LIN {X 0,Y 256.898,Z 678.395,A -85,B 0,C 180,E1 -18633.136,E2 -18633.136} C_VEL
LIN {X 0,Y 257.218,Z 676.163,A -85,B 0,C 180,E1 -18636.274,E2 -18636.274} C_VEL
LIN {X 0,Y 258.082,Z 673.338,A -85,B 0,C 180,E1 -18638.614,E2 -18638.614} C_VEL
LIN {X 0,Y 259.211,Z 669.508,A -85,B 0,C 180,E1 -18640.94,E2 -18640.94} C_VEL
LIN {X 0,Y 260.376,Z 664.426,A -85,B 0,C 180,E1 -18643.342,E2 -18643.342} C_VEL
LIN {X 0,Y 261.879,Z 658.391,A -85,B 0,C 180,E1 -18645.567,E2 -18645.567} C_VEL
LIN {X 0,Y 263.703,Z 650.606,A -85,B 0,C 180,E1 -18647.847,E2 -18647.847} C_VEL
LIN {X 0,Y 265.636,Z 640.929,A -85,B 0,C 180,E1 -18650.117,E2 -18650.117} C_VEL
LIN {X 0,Y 267.345,Z 631.877,A -85,B 0,C 180,E1 -18651.796,E2 -18651.796} C_VEL
LIN {X 0,Y 269.137,Z 621.362,A -85,B 0,C 180,E1 -18653.355,E2 -18653.355} C_VEL
LIN {X 0,Y 270.675,Z 609.83,A -85,B 0,C 180,E1 -18654.712,E2 -18654.712} C_VEL
LIN {X 0,Y 271.973,Z 598.532,A -85,B 0,C 180,E1 -18655.719,E2 -18655.719} C_VEL
LIN {X 0,Y 272.565,Z 586.357,A -85,B 0,C 180,E1 -18656.554,E2 -18656.554} C_VEL
LIN {X 0,Y 272.931,Z 573.758,A -85,B 0,C 180,E1 -18657.114,E2 -18657.114} C_VEL
LIN {X 0,Y 273.749,Z 534.07,A -85,B 0,C 180,E1 -18658.199,E2 -18658.199} C_VEL
LIN {X 0,Y 273.781,Z 527.785,A -85,B 0,C 180,E1 -18658.381,E2 -18658.381} C_VEL
LIN {X 0,Y 266.212,Z 511.696,A -85,B 0,C 180,E1 -18659.794,E2 -18659.794} C_VEL
LIN {X 0,Y 257.73,Z 496.288,A -85,B 0,C 180,E1 -18661.42,E2 -18661.42} C_VEL
LIN {X 0,Y 256.336,Z 493.738,A -85,B 0,C 180,E1 -18661.726,E2 -18661.726} C_VEL
LIN {X 0,Y 256.105,Z 492.716,A -85,B 0,C 180,E1 -18662.044,E2 -18662.044} C_VEL
LIN {X 0,Y 256.108,Z 492.575,A -85,B 0,C 180,E1 -18665.188,E2 -18665.188} C_VEL
LIN {X 0,Y 256.071,Z 492.587,A -85,B 0,C 180,E1 -18669.141,E2 -18669.141} C_VEL
LIN {X 0,Y 256.063,Z 492.56,A -85,B 0,C 180,E1 -18673.326,E2 -18673.326} C_VEL
LIN {X 0,Y 256.07,Z 492.567,A -85,B 0,C 180,E1 -18677.818,E2 -18677.818} C_VEL
LIN {X 0,Y 256.068,Z 492.545,A -85,B 0,C 180,E1 -18680.857,E2 -18680.857} C_VEL
LIN {X 0,Y 256.126,Z 492.571,A -85,B 0,C 180,E1 -18682.866,E2 -18682.866} C_VEL
LIN {X 0,Y 256.064,Z 492.561,A -85,B 0,C 180,E1 -18686.706,E2 -18686.706} C_VEL
LIN {X 0,Y 256.1,Z 492.529,A -85,B 0,C 180,E1 -18690.398,E2 -18690.398} C_VEL
LIN {X 0,Y 256.166,Z 492.577,A -85,B 0,C 180,E1 -18694.869,E2 -18694.869} C_VEL
LIN {X 0,Y 256.157,Z 492.568,A -85,B 0,C 180,E1 -18699.104,E2 -18699.104} C_VEL
LIN {X 0,Y 256.274,Z 492.543,A -85,B 0,C 180,E1 -18704.083,E2 -18704.083} C_VEL
LIN {X 0,Y 256.304,Z 492.547,A -85,B 0,C 180,E1 -18708.934,E2 -18708.934} C_VEL
LIN {X 0,Y 256.534,Z 492.518,A -85,B 0,C 180,E1 -18712.127,E2 -18712.127} C_VEL
LIN {X 0,Y 256.709,Z 492.489,A -85,B 0,C 180,E1 -18718.431,E2 -18718.431} C_VEL
LIN {X 0,Y 256.709,Z 492.502,A -85,B 0,C 180,E1 -18721.569,E2 -18721.569} C_VEL
LIN {X 0,Y 256.477,Z 492.531,A -85,B 0,C 180,E1 -18726.293,E2 -18726.293} C_VEL
LIN {X 0,Y 256.434,Z 492.532,A -85,B 0,C 180,E1 -18728.964,E2 -18728.964} C_VEL
LIN {X 0,Y 255.721,Z 492.619,A -85,B 0,C 180,E1 -18730.273,E2 -18730.273} C_VEL
LIN {X 0,Y 252.761,Z 492.991,A -85,B 0,C 180,E1 -18732.404,E2 -18732.404} C_VEL
LIN {X 0,Y 250.289,Z 493.308,A -85,B 0,C 180,E1 -18734.139,E2 -18734.139} C_VEL
LIN {X 0,Y 249.269,Z 493.429,A -85,B 0,C 180,E1 -18735.487,E2 -18735.487} C_VEL
LIN {X 0,Y 249.207,Z 493.429,A -85,B 0,C 180,E1 -18735.944,E2 -18735.944} C_VEL
LIN {X 0,Y 249.102,Z 493.418,A -85,B 0,C 180,E1 -18739.789,E2 -18739.789} C_VEL
LIN {X 0,Y 249.147,Z 493.434,A -85,B 0,C 180,E1 -18745.032,E2 -18745.032} C_VEL
LIN {X 0,Y 249.079,Z 493.45,A -85,B 0,C 180,E1 -18748.994,E2 -18748.994} C_VEL
LIN {X 0,Y 249.027,Z 493.446,A -85,B 0,C 180,E1 -18752.426,E2 -18752.426} C_VEL
LIN {X 0,Y 249.049,Z 493.462,A -85,B 0,C 180,E1 -18756.342,E2 -18756.342} C_VEL
LIN {X 0,Y 249.003,Z 493.47,A -85,B 0,C 180,E1 -18760.479,E2 -18760.479} C_VEL
LIN {X 0,Y 249.065,Z 493.617,A -85,B 0,C 180,E1 -18764.83,E2 -18764.83} C_VEL
LIN {X 0,Y 251.785,Z 503.076,A -85,B 0,C 180,E1 -18768.346,E2 -18768.346} C_VEL
LIN {X 0,Y 254.298,Z 513.073,A -85,B 0,C 180,E1 -18771.759,E2 -18771.759} C_VEL
LIN {X 0,Y 256.079,Z 521.057,A -85,B 0,C 180,E1 -18774.325,E2 -18774.325} C_VEL
LIN {X 0,Y 257.657,Z 529.601,A -85,B 0,C 180,E1 -18776.94,E2 -18776.94} C_VEL
LIN {X 0,Y 257.297,Z 532.64,A -85,B 0,C 180,E1 -18777.708,E2 -18777.708} C_VEL
LIN {X 0,Y 261.354,Z 564.078,A -85,B 0,C 180,E1 -18779.275,E2 -18779.275} C_VEL
LIN {X 0,Y 264.389,Z 595.733,A -85,B 0,C 180,E1 -18780.613,E2 -18780.613} C_VEL
LIN {X 0,Y 265.308,Z 609.441,A -85,B 0,C 180,E1 -18781.132,E2 -18781.132} C_VEL
LIN {X 0,Y 263.989,Z 644.739,A -85,B 0,C 180,E1 -18782.096,E2 -18782.096} C_VEL
LIN {X 0,Y 262.828,Z 658.786,A -85,B 0,C 180,E1 -18782.789,E2 -18782.789} C_VEL
LIN {X 0,Y 261.25,Z 671.74,A -85,B 0,C 180,E1 -18783.757,E2 -18783.757} C_VEL
LIN {X 0,Y 259.131,Z 683.47,A -85,B 0,C 180,E1 -18784.928,E2 -18784.928} C_VEL
LIN {X 0,Y 256.83,Z 694.835,A -85,B 0,C 180,E1 -18786.41,E2 -18786.41} C_VEL
LIN {X 0,Y 254.641,Z 705.126,A -85,B 0,C 180,E1 -18788.125,E2 -18788.125} C_VEL
LIN {X 0,Y 252.582,Z 714.429,A -85,B 0,C 180,E1 -18790.072,E2 -18790.072} C_VEL
LIN {X 0,Y 250.959,Z 722.161,A -85,B 0,C 180,E1 -18792.059,E2 -18792.059} C_VEL
LIN {X 0,Y 249.69,Z 727.412,A -85,B 0,C 180,E1 -18793.653,E2 -18793.653} C_VEL
LIN {X 0,Y 248.633,Z 734.063,A -85,B 0,C 180,E1 -18796.098,E2 -18796.098} C_VEL
LIN {X 0,Y 247.979,Z 739.385,A -85,B 0,C 180,E1 -18798.558,E2 -18798.558} C_VEL
LIN {X 0,Y 247.814,Z 743.573,A -85,B 0,C 180,E1 -18801.027,E2 -18801.027} C_VEL
LIN {X 0,Y 247.978,Z 746.708,A -85,B 0,C 180,E1 -18803.491,E2 -18803.491} C_VEL
LIN {X 0,Y 248.246,Z 748.229,A -85,B 0,C 180,E1 -18805.128,E2 -18805.128} C_VEL
LIN {X 0,Y 248.493,Z 749.321,A -85,B 0,C 180,E1 -18806.757,E2 -18806.757} C_VEL
LIN {X 0,Y 248.802,Z 750.008,A -85,B 0,C 180,E1 -18808.381,E2 -18808.381} C_VEL
LIN {X 0,Y 249.233,Z 750.293,A -85,B 0,C 180,E1 -18810,E2 -18810} C_VEL
LIN {X 0,Y 248.804,Z 750,A -85,B 0,C 180,E1 -18811.619,E2 -18811.619} C_VEL
LIN {X 0,Y 248.498,Z 749.308,A -85,B 0,C 180,E1 -18813.243,E2 -18813.243} C_VEL
LIN {X 0,Y 248.261,Z 748.212,A -85,B 0,C 180,E1 -18814.872,E2 -18814.872} C_VEL
LIN {X 0,Y 247.947,Z 745.853,A -85,B 0,C 180,E1 -18817.221,E2 -18817.221} C_VEL
LIN {X 0,Y 247.818,Z 742.225,A -85,B 0,C 180,E1 -18819.797,E2 -18819.797} C_VEL
LIN {X 0,Y 248.151,Z 737.656,A -85,B 0,C 180,E1 -18822.263,E2 -18822.263} C_VEL
LIN {X 0,Y 248.949,Z 731.901,A -85,B 0,C 180,E1 -18824.718,E2 -18824.718} C_VEL
LIN {X 0,Y 250.399,Z 724.287,A -85,B 0,C 180,E1 -18827.299,E2 -18827.299} C_VEL
LIN {X 0,Y 252.186,Z 715.948,A -85,B 0,C 180,E1 -18829.537,E2 -18829.537} C_VEL
LIN {X 0,Y 254.191,Z 706.941,A -85,B 0,C 180,E1 -18831.49,E2 -18831.49} C_VEL
LIN {X 0,Y 256.635,Z 695.91,A -85,B 0,C 180,E1 -18833.395,E2 -18833.395} C_VEL
LIN {X 0,Y 258.839,Z 684.792,A -85,B 0,C 180,E1 -18834.888,E2 -18834.888} C_VEL
LIN {X 0,Y 261.021,Z 672.375,A -85,B 0,C 180,E1 -18836.16,E2 -18836.16} C_VEL
LIN {X 0,Y 262.652,Z 659.498,A -85,B 0,C 180,E1 -18837.141,E2 -18837.141} C_VEL
LIN {X 0,Y 263.825,Z 646.314,A -85,B 0,C 180,E1 -18837.81,E2 -18837.81} C_VEL
LIN {X 0,Y 264.634,Z 624.724,A -85,B 0,C 180,E1 -18838.448,E2 -18838.448} C_VEL
LIN {X 0,Y 265.119,Z 606.949,A -85,B 0,C 180,E1 -18838.926,E2 -18838.926} C_VEL
LIN {X 0,Y 262.716,Z 577.983,A -85,B 0,C 180,E1 -18840.087,E2 -18840.087} C_VEL
LIN {X 0,Y 259.668,Z 550.828,A -85,B 0,C 180,E1 -18841.31,E2 -18841.31} C_VEL
LIN {X 0,Y 257.249,Z 532.626,A -85,B 0,C 180,E1 -18842.256,E2 -18842.256} C_VEL
LIN {X 0,Y 257.663,Z 529.472,A -85,B 0,C 180,E1 -18843.059,E2 -18843.059} C_VEL
LIN {X 0,Y 255.438,Z 518.047,A -85,B 0,C 180,E1 -18846.582,E2 -18846.582} C_VEL
LIN {X 0,Y 252.912,Z 507.399,A -85,B 0,C 180,E1 -18850.085,E2 -18850.085} C_VEL
LIN {X 0,Y 250.225,Z 497.431,A -85,B 0,C 180,E1 -18853.648,E2 -18853.648} C_VEL
LIN {X 0,Y 249.047,Z 493.501,A -85,B 0,C 180,E1 -18855.201,E2 -18855.201} C_VEL
LIN {X 0,Y 249.004,Z 493.47,A -85,B 0,C 180,E1 -18859.644,E2 -18859.644} C_VEL
LIN {X 0,Y 249.044,Z 493.462,A -85,B 0,C 180,E1 -18863.657,E2 -18863.657} C_VEL
LIN {X 0,Y 249.033,Z 493.449,A -85,B 0,C 180,E1 -18867.845,E2 -18867.845} C_VEL
LIN {X 0,Y 249.093,Z 493.441,A -85,B 0,C 180,E1 -18871.338,E2 -18871.338} C_VEL
LIN {X 0,Y 249.147,Z 493.435,A -85,B 0,C 180,E1 -18874.968,E2 -18874.968} C_VEL
LIN {X 0,Y 249.102,Z 493.417,A -85,B 0,C 180,E1 -18880.211,E2 -18880.211} C_VEL
LIN {X 0,Y 249.237,Z 493.425,A -85,B 0,C 180,E1 -18883.622,E2 -18883.622} C_VEL
LIN {X 0,Y 249.239,Z 493.419,A -85,B 0,C 180,E1 -18888.616,E2 -18888.616} C_VEL
LIN {X 0,Y 249.449,Z 493.411,A -85,B 0,C 180,E1 -18891.902,E2 -18891.902} C_VEL
LIN {X 0,Y 249.292,Z 493.41,A -85,B 0,C 180,E1 -18895.148,E2 -18895.148} C_VEL
LIN {X 0,Y 249.671,Z 493.382,A -85,B 0,C 180,E1 -18898.387,E2 -18898.387} C_VEL
LIN {X 0,Y 249.671,Z 493.368,A -85,B 0,C 180,E1 -18901.613,E2 -18901.613} C_VEL
LIN {X 0,Y 249.437,Z 493.41,A -85,B 0,C 180,E1 -18906.709,E2 -18906.709} C_VEL
LIN {X 0,Y 249.338,Z 493.403,A -85,B 0,C 180,E1 -18909.737,E2 -18909.737} C_VEL
LIN {X 0,Y 249.192,Z 493.432,A -85,B 0,C 180,E1 -18914.704,E2 -18914.704} C_VEL
LIN {X 0,Y 249.129,Z 493.447,A -85,B 0,C 180,E1 -18918.078,E2 -18918.078} C_VEL
LIN {X 0,Y 249.08,Z 493.444,A -85,B 0,C 180,E1 -18921.519,E2 -18921.519} C_VEL
LIN {X 0,Y 249.113,Z 493.454,A -85,B 0,C 180,E1 -18925.476,E2 -18925.476} C_VEL
LIN {X 0,Y 249.07,Z 493.412,A -85,B 0,C 180,E1 -18928.99,E2 -18928.99} C_VEL
LIN {X 0,Y 249.027,Z 493.417,A -85,B 0,C 180,E1 -18932.427,E2 -18932.427} C_VEL
LIN {X 0,Y 249.044,Z 493.463,A -85,B 0,C 180,E1 -18936.343,E2 -18936.343} C_VEL
LIN {X 0,Y 248.989,Z 493.424,A -85,B 0,C 180,E1 -18940.482,E2 -18940.482} C_VEL
LIN {X 0,Y 249.009,Z 493.456,A -85,B 0,C 180,E1 -18942.794,E2 -18942.794} C_VEL
LIN {X 0,Y 249.016,Z 493.434,A -85,B 0,C 180,E1 -18947.364,E2 -18947.364} C_VEL
LIN {X 0,Y 249.025,Z 493.447,A -85,B 0,C 180,E1 -18951.62,E2 -18951.62} C_VEL
LIN {X 0,Y 249.043,Z 493.376,A -85,B 0,C 180,E1 -18955.64,E2 -18955.64} C_VEL
LIN {X 0,Y 249.076,Z 493.63,A -85,B 0,C 180,E1 -18957.103,E2 -18957.103} C_VEL
LIN {X 0,Y 249.366,Z 494.727,A -85,B 0,C 180,E1 -18957.422,E2 -18957.422} C_VEL
LIN {X 0,Y 258.488,Z 511.081,A -85,B 0,C 180,E1 -18959.298,E2 -18959.298} C_VEL
LIN {X 0,Y 265.326,Z 524.858,A -85,B 0,C 180,E1 -18960.631,E2 -18960.631} C_VEL
LIN {X 0,Y 267.603,Z 530.043,A -85,B 0,C 180,E1 -18961.073,E2 -18961.073} C_VEL
LIN {X 0,Y 266.729,Z 570.85,A -85,B 0,C 180,E1 -18962.201,E2 -18962.201} C_VEL
LIN {X 0,Y 266.366,Z 584.382,A -85,B 0,C 180,E1 -18962.736,E2 -18962.736} C_VEL
LIN {X 0,Y 265.506,Z 597.64,A -85,B 0,C 180,E1 -18963.576,E2 -18963.576} C_VEL
LIN {X 0,Y 264.349,Z 609.929,A -85,B 0,C 180,E1 -18964.68,E2 -18964.68} C_VEL
LIN {X 0,Y 262.733,Z 621.407,A -85,B 0,C 180,E1 -18966.03,E2 -18966.03} C_VEL
LIN {X 0,Y 260.875,Z 632.144,A -85,B 0,C 180,E1 -18967.634,E2 -18967.634} C_VEL
LIN {X 0,Y 259.092,Z 641.336,A -85,B 0,C 180,E1 -18969.352,E2 -18969.352} C_VEL
LIN {X 0,Y 257.375,Z 649.686,A -85,B 0,C 180,E1 -18971.286,E2 -18971.286} C_VEL
LIN {X 0,Y 255.459,Z 657.796,A -85,B 0,C 180,E1 -18973.621,E2 -18973.621} C_VEL
LIN {X 0,Y 253.631,Z 664.903,A -85,B 0,C 180,E1 -18976.21,E2 -18976.21} C_VEL
LIN {X 0,Y 252.34,Z 670.272,A -85,B 0,C 180,E1 -18978.758,E2 -18978.758} C_VEL
LIN {X 0,Y 251.142,Z 674.161,A -85,B 0,C 180,E1 -18981.146,E2 -18981.146} C_VEL
LIN {X 0,Y 250.245,Z 677.03,A -85,B 0,C 180,E1 -18983.55,E2 -18983.55} C_VEL
LIN {X 0,Y 250.031,Z 678.371,A -85,B 0,C 180,E1 -18985.163,E2 -18985.163} C_VEL
LIN {X 0,Y 249.892,Z 679.322,A -85,B 0,C 180,E1 -18986.776,E2 -18986.776} C_VEL
LIN {X 0,Y 249.637,Z 680.15,A -85,B 0,C 180,E1 -18990,E2 -18990} C_VEL
LIN {X 0,Y 249.886,Z 679.382,A -85,B 0,C 180,E1 -18993.224,E2 -18993.224} C_VEL
LIN {X 0,Y 250.23,Z 677.151,A -85,B 0,C 180,E1 -18996.45,E2 -18996.45} C_VEL
LIN {X 0,Y 251.135,Z 674.326,A -85,B 0,C 180,E1 -18998.854,E2 -18998.854} C_VEL
LIN {X 0,Y 252.315,Z 670.495,A -85,B 0,C 180,E1 -19001.243,E2 -19001.243} C_VEL
LIN {X 0,Y 253.543,Z 665.412,A -85,B 0,C 180,E1 -19003.709,E2 -19003.709} C_VEL
LIN {X 0,Y 255.116,Z 659.377,A -85,B 0,C 180,E1 -19005.99,E2 -19005.99} C_VEL
LIN {X 0,Y 257.022,Z 651.591,A -85,B 0,C 180,E1 -19008.327,E2 -19008.327} C_VEL
LIN {X 0,Y 259.046,Z 641.914,A -85,B 0,C 180,E1 -19010.652,E2 -19010.652} C_VEL
LIN {X 0,Y 260.832,Z 632.861,A -85,B 0,C 180,E1 -19012.37,E2 -19012.37} C_VEL
LIN {X 0,Y 262.707,Z 622.343,A -85,B 0,C 180,E1 -19013.962,E2 -19013.962} C_VEL
LIN {X 0,Y 264.337,Z 610.656,A -85,B 0,C 180,E1 -19015.364,E2 -19015.364} C_VEL
LIN {X 0,Y 265.692,Z 599.17,A -85,B 0,C 180,E1 -19016.404,E2 -19016.404} C_VEL
LIN {X 0,Y 266.302,Z 586.905,A -85,B 0,C 180,E1 -19017.255,E2 -19017.255} C_VEL
LIN {X 0,Y 266.689,Z 574.464,A -85,B 0,C 180,E1 -19017.812,E2 -19017.812} C_VEL
LIN {X 0,Y 267.614,Z 533.588,A -85,B 0,C 180,E1 -19018.95,E2 -19018.95} C_VEL
LIN {X 0,Y 267.551,Z 529.88,A -85,B 0,C 180,E1 -19019.07,E2 -19019.07} C_VEL
LIN {X 0,Y 260.867,Z 515.53,A -85,B 0,C 180,E1 -19020.374,E2 -19020.374} C_VEL
LIN {X 0,Y 252.628,Z 500.555,A -85,B 0,C 180,E1 -19022.015,E2 -19022.015} C_VEL
LIN {X 0,Y 249.227,Z 494.41,A -85,B 0,C 180,E1 -19022.773,E2 -19022.773} C_VEL
LIN {X 0,Y 249.067,Z 493.538,A -85,B 0,C 180,E1 -19023.128,E2 -19023.128} C_VEL
LIN {X 0,Y 249.056,Z 493.44,A -85,B 0,C 180,E1 -19026.34,E2 -19026.34} C_VEL
LIN {X 0,Y 249.005,Z 493.46,A -85,B 0,C 180,E1 -19030.477,E2 -19030.477} C_VEL
LIN {X 0,Y 249.005,Z 493.459,A -85,B 0,C 180,E1 -19034.877,E2 -19034.877} C_VEL
LIN {X 0,Y 249.016,Z 493.455,A -85,B 0,C 180,E1 -19037.362,E2 -19037.362} C_VEL
LIN {X 0,Y 249.04,Z 493.438,A -85,B 0,C 180,E1 -19042.2,E2 -19042.2} C_VEL
LIN {X 0,Y 249.04,Z 493.456,A -85,B 0,C 180,E1 -19045.639,E2 -19045.639} C_VEL
LIN {X 0,Y 249.044,Z 493.401,A -85,B 0,C 180,E1 -19049.472,E2 -19049.472} C_VEL
LIN {X 0,Y 249.065,Z 493.451,A -85,B 0,C 180,E1 -19053.161,E2 -19053.161} C_VEL
LIN {X 0,Y 249.057,Z 493.448,A -85,B 0,C 180,E1 -19056.73,E2 -19056.73} C_VEL
LIN {X 0,Y 249.103,Z 493.455,A -85,B 0,C 180,E1 -19060.211,E2 -19060.211} C_VEL
LIN {X 0,Y 249.218,Z 493.421,A -85,B 0,C 180,E1 -19063.62,E2 -19063.62} C_VEL
LIN {X 0,Y 249.247,Z 493.43,A -85,B 0,C 180,E1 -19068.616,E2 -19068.616} C_VEL
LIN {X 0,Y 249.476,Z 493.394,A -85,B 0,C 180,E1 -19071.903,E2 -19071.903} C_VEL
LIN {X 0,Y 249.43,Z 493.392,A -85,B 0,C 180,E1 -19076.769,E2 -19076.769} C_VEL
LIN {X 0,Y 249.73,Z 493.374,A -85,B 0,C 180,E1 -19080,E2 -19080} C_VEL
LIN {X 0,Y 249.43,Z 493.394,A -85,B 0,C 180,E1 -19083.23,E2 -19083.23} C_VEL
LIN {X 0,Y 249.449,Z 493.408,A -85,B 0,C 180,E1 -19086.471,E2 -19086.471} C_VEL
LIN {X 0,Y 249.338,Z 493.411,A -85,B 0,C 180,E1 -19089.737,E2 -19089.737} C_VEL
LIN {X 0,Y 249.2,Z 493.443,A -85,B 0,C 180,E1 -19094.704,E2 -19094.704} C_VEL
LIN {X 0,Y 249.207,Z 493.429,A -85,B 0,C 180,E1 -19095.944,E2 -19095.944} C_VEL
LIN {X 0,Y 248.922,Z 493.461,A -85,B 0,C 180,E1 -19096.846,E2 -19096.846} C_VEL
LIN {X 0,Y 247.565,Z 493.63,A -85,B 0,C 180,E1 -19098.177,E2 -19098.177} C_VEL
LIN {X 0,Y 243.13,Z 494.189,A -85,B 0,C 180,E1 -19101.276,E2 -19101.276} C_VEL
LIN {X 0,Y 242.074,Z 494.331,A -85,B 0,C 180,E1 -19102.667,E2 -19102.667} C_VEL
LIN {X 0,Y 242.001,Z 494.333,A -85,B 0,C 180,E1 -19103.138,E2 -19103.138} C_VEL
LIN {X 0,Y 242.063,Z 494.306,A -85,B 0,C 180,E1 -19105.839,E2 -19105.839} C_VEL
LIN {X 0,Y 242.026,Z 494.335,A -85,B 0,C 180,E1 -19109.581,E2 -19109.581} C_VEL
LIN {X 0,Y 241.978,Z 494.322,A -85,B 0,C 180,E1 -19113.493,E2 -19113.493} C_VEL
LIN {X 0,Y 241.989,Z 494.328,A -85,B 0,C 180,E1 -19117.582,E2 -19117.582} C_VEL
LIN {X 0,Y 241.937,Z 494.32,A -85,B 0,C 180,E1 -19121.922,E2 -19121.922} C_VEL
LIN {X 0,Y 242.017,Z 494.458,A -85,B 0,C 180,E1 -19123.847,E2 -19123.847} C_VEL
LIN {X 0,Y 244.866,Z 504.204,A -85,B 0,C 180,E1 -19127.651,E2 -19127.651} C_VEL
LIN {X 0,Y 247.701,Z 515.638,A -85,B 0,C 180,E1 -19131.686,E2 -19131.686} C_VEL
LIN {X 0,Y 249.66,Z 524.87,A -85,B 0,C 180,E1 -19134.722,E2 -19134.722} C_VEL
LIN {X 0,Y 250.846,Z 531.586,A -85,B 0,C 180,E1 -19136.772,E2 -19136.772} C_VEL
LIN {X 0,Y 253.162,Z 548.651,A -85,B 0,C 180,E1 -19137.709,E2 -19137.709} C_VEL
LIN {X 0,Y 256.382,Z 576.607,A -85,B 0,C 180,E1 -19139.036,E2 -19139.036} C_VEL
LIN {X 0,Y 258.761,Z 604.007,A -85,B 0,C 180,E1 -19140.193,E2 -19140.193} C_VEL
LIN {X 0,Y 258.961,Z 611.982,A -85,B 0,C 180,E1 -19140.465,E2 -19140.465} C_VEL
LIN {X 0,Y 257.728,Z 643.741,A -85,B 0,C 180,E1 -19141.355,E2 -19141.355} C_VEL
LIN {X 0,Y 256.581,Z 657.306,A -85,B 0,C 180,E1 -19142.034,E2 -19142.034} C_VEL
LIN {X 0,Y 255.017,Z 669.723,A -85,B 0,C 180,E1 -19142.954,E2 -19142.954} C_VEL
LIN {X 0,Y 253.055,Z 680.888,A -85,B 0,C 180,E1 -19144.061,E2 -19144.061} C_VEL
LIN {X 0,Y 250.628,Z 692.538,A -85,B 0,C 180,E1 -19145.569,E2 -19145.569} C_VEL
LIN {X 0,Y 248.24,Z 703.065,A -85,B 0,C 180,E1 -19147.311,E2 -19147.311} C_VEL
LIN {X 0,Y 246.28,Z 711.721,A -85,B 0,C 180,E1 -19149.102,E2 -19149.102} C_VEL
LIN {X 0,Y 244.463,Z 719.745,A -85,B 0,C 180,E1 -19151.13,E2 -19151.13} C_VEL
LIN {X 0,Y 242.599,Z 727.604,A -85,B 0,C 180,E1 -19153.594,E2 -19153.594} C_VEL
LIN {X 0,Y 241.379,Z 734.947,A -85,B 0,C 180,E1 -19156.531,E2 -19156.531} C_VEL
LIN {X 0,Y 240.814,Z 739.88,A -85,B 0,C 180,E1 -19159.065,E2 -19159.065} C_VEL
LIN {X 0,Y 240.762,Z 743.709,A -85,B 0,C 180,E1 -19161.608,E2 -19161.608} C_VEL
LIN {X 0,Y 240.915,Z 745.709,A -85,B 0,C 180,E1 -19163.299,E2 -19163.299} C_VEL
LIN {X 0,Y 241.157,Z 747.229,A -85,B 0,C 180,E1 -19164.984,E2 -19164.984} C_VEL
LIN {X 0,Y 241.433,Z 748.327,A -85,B 0,C 180,E1 -19166.662,E2 -19166.662} C_VEL
LIN {X 0,Y 241.741,Z 749.015,A -85,B 0,C 180,E1 -19168.334,E2 -19168.334} C_VEL
LIN {X 0,Y 242.193,Z 749.304,A -85,B 0,C 180,E1 -19170,E2 -19170} C_VEL
LIN {X 0,Y 241.438,Z 748.313,A -85,B 0,C 180,E1 -19173.337,E2 -19173.337} C_VEL
LIN {X 0,Y 241.194,Z 747.214,A -85,B 0,C 180,E1 -19175.015,E2 -19175.015} C_VEL
LIN {X 0,Y 240.874,Z 745.069,A -85,B 0,C 180,E1 -19177.241,E2 -19177.241} C_VEL
LIN {X 0,Y 240.772,Z 741.218,A -85,B 0,C 180,E1 -19180.086,E2 -19180.086} C_VEL
LIN {X 0,Y 241.139,Z 736.645,A -85,B 0,C 180,E1 -19182.626,E2 -19182.626} C_VEL
LIN {X 0,Y 242.025,Z 730.892,A -85,B 0,C 180,E1 -19185.15,E2 -19185.15} C_VEL
LIN {X 0,Y 243.427,Z 723.996,A -85,B 0,C 180,E1 -19187.573,E2 -19187.573} C_VEL
LIN {X 0,Y 245.094,Z 716.568,A -85,B 0,C 180,E1 -19189.689,E2 -19189.689} C_VEL
LIN {X 0,Y 247.115,Z 707.915,A -85,B 0,C 180,E1 -19191.698,E2 -19191.698} C_VEL
LIN {X 0,Y 249.579,Z 697.284,A -85,B 0,C 180,E1 -19193.657,E2 -19193.657} C_VEL
LIN {X 0,Y 252.099,Z 685.354,A -85,B 0,C 180,E1 -19195.38,E2 -19195.38} C_VEL
LIN {X 0,Y 254.357,Z 673.372,A -85,B 0,C 180,E1 -19196.679,E2 -19196.679} C_VEL
LIN {X 0,Y 256.057,Z 660.894,A -85,B 0,C 180,E1 -19197.702,E2 -19197.702} C_VEL
LIN {X 0,Y 257.397,Z 647.822,A -85,B 0,C 180,E1 -19198.444,E2 -19198.444} C_VEL
LIN {X 0,Y 258.167,Z 633.463,A -85,B 0,C 180,E1 -19198.926,E2 -19198.926} C_VEL
LIN {X 0,Y 258.835,Z 606.75,A -85,B 0,C 180,E1 -19199.671,E2 -19199.671} C_VEL
LIN {X 0,Y 256.405,Z 577.658,A -85,B 0,C 180,E1 -19200.885,E2 -19200.885} C_VEL
LIN {X 0,Y 253.501,Z 551.579,A -85,B 0,C 180,E1 -19202.104,E2 -19202.104} C_VEL
LIN {X 0,Y 250.827,Z 531.562,A -85,B 0,C 180,E1 -19203.188,E2 -19203.188} C_VEL
LIN {X 0,Y 250.082,Z 527.007,A -85,B 0,C 180,E1 -19204.553,E2 -19204.553} C_VEL
LIN {X 0,Y 248.156,Z 517.819,A -85,B 0,C 180,E1 -19207.535,E2 -19207.535} C_VEL
LIN {X 0,Y 245.987,Z 508.715,A -85,B 0,C 180,E1 -19210.661,E2 -19210.661} C_VEL
LIN {X 0,Y 243.679,Z 500.036,A -85,B 0,C 180,E1 -19213.86,E2 -19213.86} C_VEL
LIN {X 0,Y 242.014,Z 494.391,A -85,B 0,C 180,E1 -19216.152,E2 -19216.152} C_VEL
LIN {X 0,Y 241.953,Z 494.34,A -85,B 0,C 180,E1 -19220.28,E2 -19220.28} C_VEL
LIN {X 0,Y 241.984,Z 494.341,A -85,B 0,C 180,E1 -19224.489,E2 -19224.489} C_VEL
LIN {X 0,Y 241.971,Z 494.335,A -85,B 0,C 180,E1 -19228.479,E2 -19228.479} C_VEL
LIN {X 0,Y 242.004,Z 494.312,A -85,B 0,C 180,E1 -19232.312,E2 -19232.312} C_VEL
LIN {X 0,Y 242.052,Z 494.331,A -85,B 0,C 180,E1 -19236.015,E2 -19236.015} C_VEL
LIN {X 0,Y 242.03,Z 494.303,A -85,B 0,C 180,E1 -19239.607,E2 -19239.607} C_VEL
LIN {X 0,Y 242.159,Z 494.299,A -85,B 0,C 180,E1 -19243.278,E2 -19243.278} C_VEL
LIN {X 0,Y 242.175,Z 494.299,A -85,B 0,C 180,E1 -19248.279,E2 -19248.279} C_VEL
LIN {X 0,Y 242.395,Z 494.29,A -85,B 0,C 180,E1 -19251.665,E2 -19251.665} C_VEL
LIN {X 0,Y 242.252,Z 494.287,A -85,B 0,C 180,E1 -19255.007,E2 -19255.007} C_VEL
LIN {X 0,Y 242.631,Z 494.259,A -85,B 0,C 180,E1 -19258.34,E2 -19258.34} C_VEL
LIN {X 0,Y 242.631,Z 494.243,A -85,B 0,C 180,E1 -19261.66,E2 -19261.66} C_VEL
LIN {X 0,Y 242.418,Z 494.286,A -85,B 0,C 180,E1 -19266.681,E2 -19266.681} C_VEL
LIN {X 0,Y 242.262,Z 494.285,A -85,B 0,C 180,E1 -19270.024,E2 -19270.024} C_VEL
LIN {X 0,Y 242.151,Z 494.305,A -85,B 0,C 180,E1 -19275.142,E2 -19275.142} C_VEL
LIN {X 0,Y 242.065,Z 494.33,A -85,B 0,C 180,E1 -19278.625,E2 -19278.625} C_VEL
LIN {X 0,Y 242.002,Z 494.322,A -85,B 0,C 180,E1 -19282.181,E2 -19282.181} C_VEL
LIN {X 0,Y 242.063,Z 494.332,A -85,B 0,C 180,E1 -19285.839,E2 -19285.839} C_VEL
LIN {X 0,Y 242.004,Z 494.282,A -85,B 0,C 180,E1 -19289.584,E2 -19289.584} C_VEL
LIN {X 0,Y 241.977,Z 494.315,A -85,B 0,C 180,E1 -19293.493,E2 -19293.493} C_VEL
LIN {X 0,Y 241.986,Z 494.322,A -85,B 0,C 180,E1 -19297.583,E2 -19297.583} C_VEL
LIN {X 0,Y 241.933,Z 494.317,A -85,B 0,C 180,E1 -19301.924,E2 -19301.924} C_VEL
LIN {X 0,Y 241.935,Z 494.318,A -85,B 0,C 180,E1 -19306.572,E2 -19306.572} C_VEL
LIN {X 0,Y 241.955,Z 494.347,A -85,B 0,C 180,E1 -19310.282,E2 -19310.282} C_VEL
LIN {X 0,Y 241.981,Z 494.258,A -85,B 0,C 180,E1 -19314.489,E2 -19314.489} C_VEL
LIN {X 0,Y 242.053,Z 494.601,A -85,B 0,C 180,E1 -19316.082,E2 -19316.082} C_VEL
LIN {X 0,Y 242.36,Z 495.793,A -85,B 0,C 180,E1 -19316.359,E2 -19316.359} C_VEL
LIN {X 0,Y 251.819,Z 512.356,A -85,B 0,C 180,E1 -19318.398,E2 -19318.398} C_VEL
LIN {X 0,Y 259.348,Z 527.313,A -85,B 0,C 180,E1 -19319.931,E2 -19319.931} C_VEL
LIN {X 0,Y 261.396,Z 532.057,A -85,B 0,C 180,E1 -19320.35,E2 -19320.35} C_VEL
LIN {X 0,Y 260.534,Z 573.012,A -85,B 0,C 180,E1 -19321.516,E2 -19321.516} C_VEL
LIN {X 0,Y 260.13,Z 586.272,A -85,B 0,C 180,E1 -19322.08,E2 -19322.08} C_VEL
LIN {X 0,Y 259.225,Z 598.638,A -85,B 0,C 180,E1 -19322.884,E2 -19322.884} C_VEL
LIN {X 0,Y 258.014,Z 610.923,A -85,B 0,C 180,E1 -19324.012,E2 -19324.012} C_VEL
LIN {X 0,Y 256.332,Z 622.398,A -85,B 0,C 180,E1 -19325.392,E2 -19325.392} C_VEL
LIN {X 0,Y 254.39,Z 633.136,A -85,B 0,C 180,E1 -19327.032,E2 -19327.032} C_VEL
LIN {X 0,Y 252.527,Z 642.328,A -85,B 0,C 180,E1 -19328.79,E2 -19328.79} C_VEL
LIN {X 0,Y 250.728,Z 650.677,A -85,B 0,C 180,E1 -19330.771,E2 -19330.771} C_VEL
LIN {X 0,Y 248.724,Z 658.787,A -85,B 0,C 180,E1 -19333.165,E2 -19333.165} C_VEL
LIN {X 0,Y 246.812,Z 665.893,A -85,B 0,C 180,E1 -19335.821,E2 -19335.821} C_VEL
LIN {X 0,Y 245.451,Z 671.262,A -85,B 0,C 180,E1 -19338.438,E2 -19338.438} C_VEL
LIN {X 0,Y 244.2,Z 675.15,A -85,B 0,C 180,E1 -19340.893,E2 -19340.893} C_VEL
LIN {X 0,Y 243.26,Z 678.019,A -85,B 0,C 180,E1 -19343.364,E2 -19343.364} C_VEL
LIN {X 0,Y 243.028,Z 679.36,A -85,B 0,C 180,E1 -19345.023,E2 -19345.023} C_VEL
LIN {X 0,Y 242.879,Z 680.31,A -85,B 0,C 180,E1 -19346.682,E2 -19346.682} C_VEL
LIN {X 0,Y 242.61,Z 681.138,A -85,B 0,C 180,E1 -19350,E2 -19350} C_VEL
LIN {X 0,Y 242.873,Z 680.369,A -85,B 0,C 180,E1 -19353.318,E2 -19353.318} C_VEL
LIN {X 0,Y 243.245,Z 678.138,A -85,B 0,C 180,E1 -19356.636,E2 -19356.636} C_VEL
LIN {X 0,Y 244.193,Z 675.313,A -85,B 0,C 180,E1 -19359.108,E2 -19359.108} C_VEL
LIN {X 0,Y 245.425,Z 671.482,A -85,B 0,C 180,E1 -19361.563,E2 -19361.563} C_VEL
LIN {X 0,Y 246.721,Z 666.399,A -85,B 0,C 180,E1 -19364.095,E2 -19364.095} C_VEL
LIN {X 0,Y 248.367,Z 660.363,A -85,B 0,C 180,E1 -19366.437,E2 -19366.437} C_VEL
LIN {X 0,Y 250.36,Z 652.577,A -85,B 0,C 180,E1 -19368.833,E2 -19368.833} C_VEL
LIN {X 0,Y 252.48,Z 642.9,A -85,B 0,C 180,E1 -19371.214,E2 -19371.214} C_VEL
LIN {X 0,Y 254.348,Z 633.845,A -85,B 0,C 180,E1 -19372.972,E2 -19372.972} C_VEL
LIN {X 0,Y 256.301,Z 623.326,A -85,B 0,C 180,E1 -19374.6,E2 -19374.6} C_VEL
LIN {X 0,Y 258.007,Z 611.638,A -85,B 0,C 180,E1 -19376.032,E2 -19376.032} C_VEL
LIN {X 0,Y 259.412,Z 600.151,A -85,B 0,C 180,E1 -19377.095,E2 -19377.095} C_VEL
LIN {X 0,Y 260.082,Z 587.515,A -85,B 0,C 180,E1 -19377.985,E2 -19377.985} C_VEL
LIN {X 0,Y 260.489,Z 575.314,A -85,B 0,C 180,E1 -19378.538,E2 -19378.538} C_VEL
LIN {X 0,Y 261.455,Z 534.264,A -85,B 0,C 180,E1 -19379.708,E2 -19379.708} C_VEL
LIN {X 0,Y 261.41,Z 531.937,A -85,B 0,C 180,E1 -19379.787,E2 -19379.787} C_VEL
LIN {X 0,Y 254.491,Z 517.288,A -85,B 0,C 180,E1 -19381.195,E2 -19381.195} C_VEL
LIN {X 0,Y 245.744,Z 501.586,A -85,B 0,C 180,E1 -19383.027,E2 -19383.027} C_VEL
LIN {X 0,Y 243.114,Z 497.349,A -85,B 0,C 180,E1 -19383.595,E2 -19383.595} C_VEL
LIN {X 0,Y 242.134,Z 494.974,A -85,B 0,C 180,E1 -19383.934,E2 -19383.934} C_VEL
LIN {X 0,Y 242.022,Z 494.377,A -85,B 0,C 180,E1 -19384.368,E2 -19384.368} C_VEL
LIN {X 0,Y 241.995,Z 494.327,A -85,B 0,C 180,E1 -19388.359,E2 -19388.359} C_VEL
LIN {X 0,Y 241.937,Z 494.319,A -85,B 0,C 180,E1 -19391.921,E2 -19391.921} C_VEL
LIN {X 0,Y 241.935,Z 494.349,A -85,B 0,C 180,E1 -19396.57,E2 -19396.57} C_VEL
LIN {X 0,Y 241.992,Z 494.305,A -85,B 0,C 180,E1 -19401.639,E2 -19401.639} C_VEL
LIN {X 0,Y 241.984,Z 494.343,A -85,B 0,C 180,E1 -19404.488,E2 -19404.488} C_VEL
LIN {X 0,Y 241.969,Z 494.285,A -85,B 0,C 180,E1 -19408.479,E2 -19408.479} C_VEL
LIN {X 0,Y 241.997,Z 494.315,A -85,B 0,C 180,E1 -19412.311,E2 -19412.311} C_VEL
LIN {X 0,Y 242.037,Z 494.33,A -85,B 0,C 180,E1 -19416.014,E2 -19416.014} C_VEL
LIN {X 0,Y 242.031,Z 494.332,A -85,B 0,C 180,E1 -19419.607,E2 -19419.607} C_VEL
LIN {X 0,Y 242.159,Z 494.302,A -85,B 0,C 180,E1 -19423.278,E2 -19423.278} C_VEL
LIN {X 0,Y 242.181,Z 494.314,A -85,B 0,C 180,E1 -19428.279,E2 -19428.279} C_VEL
LIN {X 0,Y 242.423,Z 494.269,A -85,B 0,C 180,E1 -19431.665,E2 -19431.665} C_VEL
LIN {X 0,Y 242.255,Z 494.302,A -85,B 0,C 180,E1 -19435.007,E2 -19435.007} C_VEL
LIN {X 0,Y 242.631,Z 494.241,A -85,B 0,C 180,E1 -19438.34,E2 -19438.34} C_VEL
LIN {X 0,Y 242.631,Z 494.255,A -85,B 0,C 180,E1 -19441.66,E2 -19441.66} C_VEL
LIN {X 0,Y 242.419,Z 494.284,A -85,B 0,C 180,E1 -19446.659,E2 -19446.659} C_VEL
LIN {X 0,Y 242.262,Z 494.29,A -85,B 0,C 180,E1 -19450.024,E2 -19450.024} C_VEL
LIN {X 0,Y 242.162,Z 494.318,A -85,B 0,C 180,E1 -19455.141,E2 -19455.141} C_VEL
LIN {X 0,Y 242.066,Z 494.289,A -85,B 0,C 180,E1 -19458.625,E2 -19458.625} C_VEL
LIN {X 0,Y 242.001,Z 494.333,A -85,B 0,C 180,E1 -19463.138,E2 -19463.138} C_VEL
LIN {X 0,Y 241.369,Z 494.415,A -85,B 0,C 180,E1 -19464.526,E2 -19464.526} C_VEL
LIN {X 0,Y 238.53,Z 494.768,A -85,B 0,C 180,E1 -19466.79,E2 -19466.79} C_VEL
LIN {X 0,Y 236.087,Z 495.073,A -85,B 0,C 180,E1 -19468.634,E2 -19468.634} C_VEL
LIN {X 0,Y 235.022,Z 495.212,A -85,B 0,C 180,E1 -19470.066,E2 -19470.066} C_VEL
LIN {X 0,Y 234.928,Z 495.222,A -85,B 0,C 180,E1 -19470.551,E2 -19470.551} C_VEL
LIN {X 0,Y 234.929,Z 495.208,A -85,B 0,C 180,E1 -19474.638,E2 -19474.638} C_VEL
LIN {X 0,Y 234.939,Z 495.207,A -85,B 0,C 180,E1 -19478.945,E2 -19478.945} C_VEL
LIN {X 0,Y 234.934,Z 495.37,A -85,B 0,C 180,E1 -19482.829,E2 -19482.829} C_VEL
LIN {X 0,Y 238.152,Z 506.239,A -85,B 0,C 180,E1 -19487.256,E2 -19487.256} C_VEL
LIN {X 0,Y 240.873,Z 517.324,A -85,B 0,C 180,E1 -19491.305,E2 -19491.305} C_VEL
LIN {X 0,Y 242.684,Z 525.743,A -85,B 0,C 180,E1 -19494.181,E2 -19494.181} C_VEL
LIN {X 0,Y 243.638,Z 530.582,A -85,B 0,C 180,E1 -19495.678,E2 -19495.678} C_VEL
LIN {X 0,Y 245.126,Z 534.825,A -85,B 0,C 180,E1 -19496.088,E2 -19496.088} C_VEL
LIN {X 0,Y 249.236,Z 567.218,A -85,B 0,C 180,E1 -19497.773,E2 -19497.773} C_VEL
LIN {X 0,Y 252.06,Z 598.456,A -85,B 0,C 180,E1 -19499.173,E2 -19499.173} C_VEL
LIN {X 0,Y 252.825,Z 610.698,A -85,B 0,C 180,E1 -19499.664,E2 -19499.664} C_VEL
LIN {X 0,Y 251.513,Z 642.794,A -85,B 0,C 180,E1 -19500.581,E2 -19500.581} C_VEL
LIN {X 0,Y 250.326,Z 656.442,A -85,B 0,C 180,E1 -19501.281,E2 -19501.281} C_VEL
LIN {X 0,Y 248.692,Z 668.728,A -85,B 0,C 180,E1 -19502.207,E2 -19502.207} C_VEL
LIN {X 0,Y 246.691,Z 679.895,A -85,B 0,C 180,E1 -19503.34,E2 -19503.34} C_VEL
LIN {X 0,Y 244.188,Z 691.544,A -85,B 0,C 180,E1 -19504.88,E2 -19504.88} C_VEL
LIN {X 0,Y 241.698,Z 702.069,A -85,B 0,C 180,E1 -19506.661,E2 -19506.661} C_VEL
LIN {X 0,Y 239.627,Z 710.72,A -85,B 0,C 180,E1 -19508.494,E2 -19508.494} C_VEL
LIN {X 0,Y 237.691,Z 718.739,A -85,B 0,C 180,E1 -19510.572,E2 -19510.572} C_VEL
LIN {X 0,Y 235.69,Z 726.591,A -85,B 0,C 180,E1 -19513.099,E2 -19513.099} C_VEL
LIN {X 0,Y 234.741,Z 732.05,A -85,B 0,C 180,E1 -19515.257,E2 -19515.257} C_VEL
LIN {X 0,Y 233.958,Z 737.373,A -85,B 0,C 180,E1 -19517.862,E2 -19517.862} C_VEL
LIN {X 0,Y 233.672,Z 741.56,A -85,B 0,C 180,E1 -19520.479,E2 -19520.479} C_VEL
LIN {X 0,Y 233.82,Z 744.705,A -85,B 0,C 180,E1 -19523.095,E2 -19523.095} C_VEL
LIN {X 0,Y 234.075,Z 746.229,A -85,B 0,C 180,E1 -19524.832,E2 -19524.832} C_VEL
LIN {X 0,Y 234.371,Z 747.333,A -85,B 0,C 180,E1 -19526.562,E2 -19526.562} C_VEL
LIN {X 0,Y 235.153,Z 748.314,A -85,B 0,C 180,E1 -19530,E2 -19530} C_VEL
LIN {X 0,Y 234.38,Z 747.319,A -85,B 0,C 180,E1 -19533.438,E2 -19533.438} C_VEL
LIN {X 0,Y 234.108,Z 746.214,A -85,B 0,C 180,E1 -19535.167,E2 -19535.167} C_VEL
LIN {X 0,Y 233.817,Z 744.25,A -85,B 0,C 180,E1 -19537.295,E2 -19537.295} C_VEL
LIN {X 0,Y 233.707,Z 740.207,A -85,B 0,C 180,E1 -19540.395,E2 -19540.395} C_VEL
LIN {X 0,Y 234.151,Z 735.636,A -85,B 0,C 180,E1 -19543.009,E2 -19543.009} C_VEL
LIN {X 0,Y 235.124,Z 729.884,A -85,B 0,C 180,E1 -19545.605,E2 -19545.605} C_VEL
LIN {X 0,Y 236.361,Z 723.986,A -85,B 0,C 180,E1 -19547.762,E2 -19547.762} C_VEL
LIN {X 0,Y 238.366,Z 715.559,A -85,B 0,C 180,E1 -19550.269,E2 -19550.269} C_VEL
LIN {X 0,Y 240.508,Z 706.91,A -85,B 0,C 180,E1 -19552.326,E2 -19552.326} C_VEL
LIN {X 0,Y 243.067,Z 696.278,A -85,B 0,C 180,E1 -19554.331,E2 -19554.331} C_VEL
LIN {X 0,Y 245.699,Z 684.35,A -85,B 0,C 180,E1 -19556.09,E2 -19556.09} C_VEL
LIN {X 0,Y 248.01,Z 672.364,A -85,B 0,C 180,E1 -19557.418,E2 -19557.418} C_VEL
LIN {X 0,Y 249.75,Z 659.881,A -85,B 0,C 180,E1 -19558.464,E2 -19558.464} C_VEL
LIN {X 0,Y 251.153,Z 646.732,A -85,B 0,C 180,E1 -19559.223,E2 -19559.223} C_VEL
LIN {X 0,Y 251.963,Z 631.717,A -85,B 0,C 180,E1 -19559.731,E2 -19559.731} C_VEL
LIN {X 0,Y 252.628,Z 607.74,A -85,B 0,C 180,E1 -19560.412,E2 -19560.412} C_VEL
LIN {X 0,Y 250.277,Z 578.587,A -85,B 0,C 180,E1 -19561.664,E2 -19561.664} C_VEL
LIN {X 0,Y 247.352,Z 551.751,A -85,B 0,C 180,E1 -19562.961,E2 -19562.961} C_VEL
LIN {X 0,Y 244.738,Z 533.577,A -85,B 0,C 180,E1 -19563.964,E2 -19563.964} C_VEL
LIN {X 0,Y 243.575,Z 530.216,A -85,B 0,C 180,E1 -19564.342,E2 -19564.342} C_VEL
LIN {X 0,Y 241.489,Z 520.121,A -85,B 0,C 180,E1 -19567.672,E2 -19567.672} C_VEL
LIN {X 0,Y 239.009,Z 509.591,A -85,B 0,C 180,E1 -19571.425,E2 -19571.425} C_VEL
LIN {X 0,Y 236.741,Z 501.451,A -85,B 0,C 180,E1 -19574.563,E2 -19574.563} C_VEL
LIN {X 0,Y 234.925,Z 495.303,A -85,B 0,C 180,E1 -19577.169,E2 -19577.169} C_VEL
LIN {X 0,Y 234.914,Z 495.208,A -85,B 0,C 180,E1 -19581.078,E2 -19581.078} C_VEL
LIN {X 0,Y 234.927,Z 495.208,A -85,B 0,C 180,E1 -19585.361,E2 -19585.361} C_VEL
LIN {X 0,Y 234.928,Z 495.222,A -85,B 0,C 180,E1 -19589.432,E2 -19589.432} C_VEL
LIN {X 0,Y 234.99,Z 495.184,A -85,B 0,C 180,E1 -19593.793,E2 -19593.793} C_VEL
LIN {X 0,Y 235.006,Z 495.187,A -85,B 0,C 180,E1 -19598.969,E2 -19598.969} C_VEL
LIN {X 0,Y 235.092,Z 495.175,A -85,B 0,C 180,E1 -19603.06,E2 -19603.06} C_VEL
LIN {X 0,Y 235.109,Z 495.182,A -85,B 0,C 180,E1 -19607.922,E2 -19607.922} C_VEL
LIN {X 0,Y 235.326,Z 495.17,A -85,B 0,C 180,E1 -19611.412,E2 -19611.412} C_VEL
LIN {X 0,Y 235.369,Z 495.163,A -85,B 0,C 180,E1 -19613.14,E2 -19613.14} C_VEL
LIN {X 0,Y 235.591,Z 495.135,A -85,B 0,C 180,E1 -19618.291,E2 -19618.291} C_VEL
LIN {X 0,Y 235.591,Z 495.119,A -85,B 0,C 180,E1 -19621.71,E2 -19621.71} C_VEL
LIN {X 0,Y 235.369,Z 495.162,A -85,B 0,C 180,E1 -19626.86,E2 -19626.86} C_VEL
LIN {X 0,Y 235.209,Z 495.165,A -85,B 0,C 180,E1 -19630.328,E2 -19630.328} C_VEL
LIN {X 0,Y 235.102,Z 495.179,A -85,B 0,C 180,E1 -19635.607,E2 -19635.607} C_VEL
LIN {X 0,Y 235.001,Z 495.213,A -85,B 0,C 180,E1 -19639.206,E2 -19639.206} C_VEL
LIN {X 0,Y 234.948,Z 495.201,A -85,B 0,C 180,E1 -19642.884,E2 -19642.884} C_VEL
LIN {X 0,Y 234.964,Z 495.209,A -85,B 0,C 180,E1 -19646.658,E2 -19646.658} C_VEL
LIN {X 0,Y 234.918,Z 495.158,A -85,B 0,C 180,E1 -19650.57,E2 -19650.57} C_VEL
LIN {X 0,Y 234.927,Z 495.215,A -85,B 0,C 180,E1 -19654.639,E2 -19654.639} C_VEL
LIN {X 0,Y 234.91,Z 495.18,A -85,B 0,C 180,E1 -19658.936,E2 -19658.936} C_VEL
LIN {X 0,Y 234.888,Z 495.224,A -85,B 0,C 180,E1 -19663.486,E2 -19663.486} C_VEL
LIN {X 0,Y 234.888,Z 495.196,A -85,B 0,C 180,E1 -19666.515,E2 -19666.515} C_VEL
LIN {X 0,Y 234.918,Z 495.216,A -85,B 0,C 180,E1 -19671.08,E2 -19671.08} C_VEL
LIN {X 0,Y 234.967,Z 495.314,A -85,B 0,C 180,E1 -19674.781,E2 -19674.781} C_VEL
LIN {X 0,Y 235.171,Z 496.249,A -85,B 0,C 180,E1 -19675.137,E2 -19675.137} C_VEL
LIN {X 0,Y 236.663,Z 498.982,A -85,B 0,C 180,E1 -19675.531,E2 -19675.531} C_VEL
LIN {X 0,Y 245.237,Z 513.641,A -85,B 0,C 180,E1 -19677.452,E2 -19677.452} C_VEL
LIN {X 0,Y 253.389,Z 529.799,A -85,B 0,C 180,E1 -19679.196,E2 -19679.196} C_VEL
LIN {X 0,Y 255.265,Z 534.083,A -85,B 0,C 180,E1 -19679.596,E2 -19679.596} C_VEL
LIN {X 0,Y 254.377,Z 573.098,A -85,B 0,C 180,E1 -19680.731,E2 -19680.731} C_VEL
LIN {X 0,Y 253.984,Z 585.841,A -85,B 0,C 180,E1 -19681.253,E2 -19681.253} C_VEL
LIN {X 0,Y 253.131,Z 598.344,A -85,B 0,C 180,E1 -19682.063,E2 -19682.063} C_VEL
LIN {X 0,Y 251.844,Z 610.897,A -85,B 0,C 180,E1 -19683.203,E2 -19683.203} C_VEL
LIN {X 0,Y 250.171,Z 622.33,A -85,B 0,C 180,E1 -19684.576,E2 -19684.576} C_VEL
LIN {X 0,Y 248.417,Z 631.817,A -85,B 0,C 180,E1 -19686.004,E2 -19686.004} C_VEL
LIN {X 0,Y 246.829,Z 639.476,A -85,B 0,C 180,E1 -19687.395,E2 -19687.395} C_VEL
LIN {X 0,Y 244.826,Z 648.509,A -85,B 0,C 180,E1 -19689.412,E2 -19689.412} C_VEL
LIN {X 0,Y 242.669,Z 657.265,A -85,B 0,C 180,E1 -19691.861,E2 -19691.861} C_VEL
LIN {X 0,Y 240.99,Z 663.438,A -85,B 0,C 180,E1 -19694.003,E2 -19694.003} C_VEL
LIN {X 0,Y 239.451,Z 669.043,A -85,B 0,C 180,E1 -19696.42,E2 -19696.42} C_VEL
LIN {X 0,Y 238.052,Z 673.651,A -85,B 0,C 180,E1 -19698.937,E2 -19698.937} C_VEL
LIN {X 0,Y 236.866,Z 677.187,A -85,B 0,C 180,E1 -19701.469,E2 -19701.469} C_VEL
LIN {X 0,Y 236.278,Z 679.008,A -85,B 0,C 180,E1 -19703.167,E2 -19703.167} C_VEL
LIN {X 0,Y 236.026,Z 680.349,A -85,B 0,C 180,E1 -19704.875,E2 -19704.875} C_VEL
LIN {X 0,Y 235.866,Z 681.298,A -85,B 0,C 180,E1 -19706.584,E2 -19706.584} C_VEL
LIN {X 0,Y 235.582,Z 682.126,A -85,B 0,C 180,E1 -19710,E2 -19710} C_VEL
LIN {X 0,Y 235.861,Z 681.357,A -85,B 0,C 180,E1 -19713.416,E2 -19713.416} C_VEL
LIN {X 0,Y 236.263,Z 679.126,A -85,B 0,C 180,E1 -19716.833,E2 -19716.833} C_VEL
LIN {X 0,Y 237.256,Z 676.3,A -85,B 0,C 180,E1 -19719.376,E2 -19719.376} C_VEL
LIN {X 0,Y 238.544,Z 672.469,A -85,B 0,C 180,E1 -19721.901,E2 -19721.901} C_VEL
LIN {X 0,Y 239.91,Z 667.385,A -85,B 0,C 180,E1 -19724.504,E2 -19724.504} C_VEL
LIN {X 0,Y 241.634,Z 661.349,A -85,B 0,C 180,E1 -19726.909,E2 -19726.909} C_VEL
LIN {X 0,Y 243.718,Z 653.563,A -85,B 0,C 180,E1 -19729.367,E2 -19729.367} C_VEL
LIN {X 0,Y 245.94,Z 643.885,A -85,B 0,C 180,E1 -19731.807,E2 -19731.807} C_VEL
LIN {X 0,Y 247.892,Z 634.83,A -85,B 0,C 180,E1 -19733.606,E2 -19733.606} C_VEL
LIN {X 0,Y 249.92,Z 624.312,A -85,B 0,C 180,E1 -19735.271,E2 -19735.271} C_VEL
LIN {X 0,Y 251.711,Z 612.62,A -85,B 0,C 180,E1 -19736.735,E2 -19736.735} C_VEL
LIN {X 0,Y 253.17,Z 601.132,A -85,B 0,C 180,E1 -19737.82,E2 -19737.82} C_VEL
LIN {X 0,Y 253.91,Z 588.8,A -85,B 0,C 180,E1 -19738.708,E2 -19738.708} C_VEL
LIN {X 0,Y 254.324,Z 575.94,A -85,B 0,C 180,E1 -19739.31,E2 -19739.31} C_VEL
LIN {X 0,Y 255.272,Z 533.889,A -85,B 0,C 180,E1 -19740.547,E2 -19740.547} C_VEL
LIN {X 0,Y 247.85,Z 518.504,A -85,B 0,C 180,E1 -19742.124,E2 -19742.124} C_VEL
LIN {X 0,Y 238.782,Z 502.542,A -85,B 0,C 180,E1 -19744.127,E2 -19744.127} C_VEL
LIN {X 0,Y 236.41,Z 498.69,A -85,B 0,C 180,E1 -19744.673,E2 -19744.673} C_VEL
LIN {X 0,Y 235.116,Z 495.964,A -85,B 0,C 180,E1 -19745.072,E2 -19745.072} C_VEL
LIN {X 0,Y 234.987,Z 495.287,A -85,B 0,C 180,E1 -19745.413,E2 -19745.413} C_VEL
LIN {X 0,Y 234.941,Z 495.214,A -85,B 0,C 180,E1 -19748.943,E2 -19748.943} C_VEL
LIN {X 0,Y 234.888,Z 495.197,A -85,B 0,C 180,E1 -19753.485,E2 -19753.485} C_VEL
LIN {X 0,Y 234.888,Z 495.227,A -85,B 0,C 180,E1 -19756.514,E2 -19756.514} C_VEL
LIN {X 0,Y 234.915,Z 495.179,A -85,B 0,C 180,E1 -19761.078,E2 -19761.078} C_VEL
LIN {X 0,Y 234.927,Z 495.216,A -85,B 0,C 180,E1 -19765.361,E2 -19765.361} C_VEL
LIN {X 0,Y 234.918,Z 495.158,A -85,B 0,C 180,E1 -19769.43,E2 -19769.43} C_VEL
LIN {X 0,Y 234.99,Z 495.21,A -85,B 0,C 180,E1 -19773.793,E2 -19773.793} C_VEL
LIN {X 0,Y 234.993,Z 495.202,A -85,B 0,C 180,E1 -19778.968,E2 -19778.968} C_VEL
LIN {X 0,Y 235.091,Z 495.183,A -85,B 0,C 180,E1 -19783.06,E2 -19783.06} C_VEL
LIN {X 0,Y 235.141,Z 495.192,A -85,B 0,C 180,E1 -19787.923,E2 -19787.923} C_VEL
LIN {X 0,Y 235.372,Z 495.144,A -85,B 0,C 180,E1 -19791.414,E2 -19791.414} C_VEL
LIN {X 0,Y 235.399,Z 495.157,A -85,B 0,C 180,E1 -19793.141,E2 -19793.141} C_VEL
LIN {X 0,Y 235.591,Z 495.117,A -85,B 0,C 180,E1 -19798.29,E2 -19798.29} C_VEL
LIN {X 0,Y 235.591,Z 495.131,A -85,B 0,C 180,E1 -19801.709,E2 -19801.709} C_VEL
LIN {X 0,Y 235.369,Z 495.162,A -85,B 0,C 180,E1 -19806.86,E2 -19806.86} C_VEL
LIN {X 0,Y 235.209,Z 495.166,A -85,B 0,C 180,E1 -19810.328,E2 -19810.328} C_VEL
LIN {X 0,Y 235.109,Z 495.192,A -85,B 0,C 180,E1 -19815.607,E2 -19815.607} C_VEL
LIN {X 0,Y 235.002,Z 495.169,A -85,B 0,C 180,E1 -19819.206,E2 -19819.206} C_VEL
LIN {X 0,Y 234.945,Z 495.216,A -85,B 0,C 180,E1 -19823.124,E2 -19823.124} C_VEL
LIN {X 0,Y 234.966,Z 495.185,A -85,B 0,C 180,E1 -19826.658,E2 -19826.658} C_VEL
LIN {X 0,Y 234.928,Z 495.222,A -85,B 0,C 180,E1 -19830.551,E2 -19830.551} C_VEL
LIN {X 0,Y 234.246,Z 495.309,A -85,B 0,C 180,E1 -19831.981,E2 -19831.981} C_VEL
LIN {X 0,Y 231.407,Z 495.657,A -85,B 0,C 180,E1 -19834.315,E2 -19834.315} C_VEL
LIN {X 0,Y 228.991,Z 495.961,A -85,B 0,C 180,E1 -19836.217,E2 -19836.217} C_VEL
LIN {X 0,Y 227.935,Z 496.078,A -85,B 0,C 180,E1 -19837.693,E2 -19837.693} C_VEL
LIN {X 0,Y 227.837,Z 496.088,A -85,B 0,C 180,E1 -19838.193,E2 -19838.193} C_VEL
LIN {X 0,Y 227.867,Z 496.292,A -85,B 0,C 180,E1 -19841.742,E2 -19841.742} C_VEL
LIN {X 0,Y 230.713,Z 505.796,A -85,B 0,C 180,E1 -19845.837,E2 -19845.837} C_VEL
LIN {X 0,Y 233.154,Z 515.092,A -85,B 0,C 180,E1 -19849.465,E2 -19849.465} C_VEL
LIN {X 0,Y 235.744,Z 526.581,A -85,B 0,C 180,E1 -19853.603,E2 -19853.603} C_VEL
LIN {X 0,Y 236.274,Z 529.34,A -85,B 0,C 180,E1 -19854.449,E2 -19854.449} C_VEL
LIN {X 0,Y 239.397,Z 537.403,A -85,B 0,C 180,E1 -19855.286,E2 -19855.286} C_VEL
LIN {X 0,Y 243.361,Z 569.807,A -85,B 0,C 180,E1 -19857.018,E2 -19857.018} C_VEL
LIN {X 0,Y 246.355,Z 604.403,A -85,B 0,C 180,E1 -19858.605,E2 -19858.605} C_VEL
LIN {X 0,Y 246.592,Z 612.294,A -85,B 0,C 180,E1 -19858.898,E2 -19858.898} C_VEL
LIN {X 0,Y 245.317,Z 641.982,A -85,B 0,C 180,E1 -19859.771,E2 -19859.771} C_VEL
LIN {X 0,Y 244.057,Z 655.576,A -85,B 0,C 180,E1 -19860.481,E2 -19860.481} C_VEL
LIN {X 0,Y 242.405,Z 667.731,A -85,B 0,C 180,E1 -19861.421,E2 -19861.421} C_VEL
LIN {X 0,Y 240.344,Z 678.898,A -85,B 0,C 180,E1 -19862.578,E2 -19862.578} C_VEL
LIN {X 0,Y 237.745,Z 690.545,A -85,B 0,C 180,E1 -19864.15,E2 -19864.15} C_VEL
LIN {X 0,Y 235.481,Z 699.994,A -85,B 0,C 180,E1 -19865.772,E2 -19865.772} C_VEL
LIN {X 0,Y 232.982,Z 709.717,A -85,B 0,C 180,E1 -19867.848,E2 -19867.848} C_VEL
LIN {X 0,Y 230.937,Z 717.732,A -85,B 0,C 180,E1 -19869.979,E2 -19869.979} C_VEL
LIN {X 0,Y 229.117,Z 724.391,A -85,B 0,C 180,E1 -19872.137,E2 -19872.137} C_VEL
LIN {X 0,Y 227.826,Z 731.045,A -85,B 0,C 180,E1 -19874.799,E2 -19874.799} C_VEL
LIN {X 0,Y 226.937,Z 736.364,A -85,B 0,C 180,E1 -19877.48,E2 -19877.48} C_VEL
LIN {X 0,Y 226.607,Z 740.553,A -85,B 0,C 180,E1 -19880.179,E2 -19880.179} C_VEL
LIN {X 0,Y 226.754,Z 743.705,A -85,B 0,C 180,E1 -19882.879,E2 -19882.879} C_VEL
LIN {X 0,Y 226.975,Z 745.228,A -85,B 0,C 180,E1 -19884.67,E2 -19884.67} C_VEL
LIN {X 0,Y 227.309,Z 746.338,A -85,B 0,C 180,E1 -19886.455,E2 -19886.455} C_VEL
LIN {X 0,Y 228.111,Z 747.324,A -85,B 0,C 180,E1 -19890,E2 -19890} C_VEL
LIN {X 0,Y 227.32,Z 746.324,A -85,B 0,C 180,E1 -19893.545,E2 -19893.545} C_VEL
LIN {X 0,Y 227.025,Z 745.213,A -85,B 0,C 180,E1 -19895.329,E2 -19895.329} C_VEL
LIN {X 0,Y 226.746,Z 743.462,A -85,B 0,C 180,E1 -19897.323,E2 -19897.323} C_VEL
LIN {X 0,Y 226.673,Z 739.2,A -85,B 0,C 180,E1 -19900.721,E2 -19900.721} C_VEL
LIN {X 0,Y 227.184,Z 734.628,A -85,B 0,C 180,E1 -19903.415,E2 -19903.415} C_VEL
LIN {X 0,Y 228.243,Z 728.876,A -85,B 0,C 180,E1 -19906.088,E2 -19906.088} C_VEL
LIN {X 0,Y 229.761,Z 722.369,A -85,B 0,C 180,E1 -19908.515,E2 -19908.515} C_VEL
LIN {X 0,Y 231.684,Z 714.554,A -85,B 0,C 180,E1 -19910.881,E2 -19910.881} C_VEL
LIN {X 0,Y 233.918,Z 705.903,A -85,B 0,C 180,E1 -19912.99,E2 -19912.99} C_VEL
LIN {X 0,Y 236.531,Z 695.264,A -85,B 0,C 180,E1 -19915.049,E2 -19915.049} C_VEL
LIN {X 0,Y 239.349,Z 683.348,A -85,B 0,C 180,E1 -19916.836,E2 -19916.836} C_VEL
LIN {X 0,Y 241.709,Z 671.356,A -85,B 0,C 180,E1 -19918.195,E2 -19918.195} C_VEL
LIN {X 0,Y 243.517,Z 658.872,A -85,B 0,C 180,E1 -19919.262,E2 -19919.262} C_VEL
LIN {X 0,Y 244.998,Z 645.741,A -85,B 0,C 180,E1 -19920.03,E2 -19920.03} C_VEL
LIN {X 0,Y 245.784,Z 630.775,A -85,B 0,C 180,E1 -19920.554,E2 -19920.554} C_VEL
LIN {X 0,Y 246.479,Z 608.517,A -85,B 0,C 180,E1 -19921.195,E2 -19921.195} C_VEL
LIN {X 0,Y 243.891,Z 575.826,A -85,B 0,C 180,E1 -19922.65,E2 -19922.65} C_VEL
LIN {X 0,Y 240.383,Z 545.459,A -85,B 0,C 180,E1 -19924.223,E2 -19924.223} C_VEL
LIN {X 0,Y 238.949,Z 535.997,A -85,B 0,C 180,E1 -19924.782,E2 -19924.782} C_VEL
LIN {X 0,Y 236.221,Z 529.098,A -85,B 0,C 180,E1 -19925.542,E2 -19925.542} C_VEL
LIN {X 0,Y 233.775,Z 517.691,A -85,B 0,C 180,E1 -19929.515,E2 -19929.515} C_VEL
LIN {X 0,Y 231.012,Z 506.81,A -85,B 0,C 180,E1 -19933.675,E2 -19933.675} C_VEL
LIN {X 0,Y 228.402,Z 498.003,A -85,B 0,C 180,E1 -19937.394,E2 -19937.394} C_VEL
LIN {X 0,Y 227.869,Z 496.194,A -85,B 0,C 180,E1 -19938.267,E2 -19938.267} C_VEL
LIN {X 0,Y 227.888,Z 496.092,A -85,B 0,C 180,E1 -19943.304,E2 -19943.304} C_VEL
LIN {X 0,Y 227.876,Z 496.078,A -85,B 0,C 180,E1 -19946.377,E2 -19946.377} C_VEL
LIN {X 0,Y 227.915,Z 496.092,A -85,B 0,C 180,E1 -19950.437,E2 -19950.437} C_VEL
LIN {X 0,Y 227.924,Z 496.069,A -85,B 0,C 180,E1 -19954.425,E2 -19954.425} C_VEL
LIN {X 0,Y 227.957,Z 496.078,A -85,B 0,C 180,E1 -19958.287,E2 -19958.287} C_VEL
LIN {X 0,Y 228.03,Z 496.05,A -85,B 0,C 180,E1 -19962.826,E2 -19962.826} C_VEL
LIN {X 0,Y 228.067,Z 496.062,A -85,B 0,C 180,E1 -19967.543,E2 -19967.543} C_VEL
LIN {X 0,Y 228.263,Z 496.047,A -85,B 0,C 180,E1 -19971.144,E2 -19971.144} C_VEL
LIN {X 0,Y 228.319,Z 496.042,A -85,B 0,C 180,E1 -19972.928,E2 -19972.928} C_VEL
LIN {X 0,Y 228.549,Z 496.012,A -85,B 0,C 180,E1 -19978.238,E2 -19978.238} C_VEL
LIN {X 0,Y 228.55,Z 495.995,A -85,B 0,C 180,E1 -19981.762,E2 -19981.762} C_VEL
LIN {X 0,Y 228.32,Z 496.039,A -85,B 0,C 180,E1 -19987.073,E2 -19987.073} C_VEL
LIN {X 0,Y 228.141,Z 496.048,A -85,B 0,C 180,E1 -19990.652,E2 -19990.652} C_VEL
LIN {X 0,Y 228.055,Z 496.068,A -85,B 0,C 180,E1 -19994.273,E2 -19994.273} C_VEL
LIN {X 0,Y 227.998,Z 496.077,A -85,B 0,C 180,E1 -19997.954,E2 -19997.954} C_VEL
LIN {X 0,Y 227.912,Z 496.076,A -85,B 0,C 180,E1 -20002.321,E2 -20002.321} C_VEL
LIN {X 0,Y 227.938,Z 496.084,A -85,B 0,C 180,E1 -20006.603,E2 -20006.603} C_VEL
LIN {X 0,Y 227.893,Z 496.032,A -85,B 0,C 180,E1 -20010.291,E2 -20010.291} C_VEL
LIN {X 0,Y 227.874,Z 496.073,A -85,B 0,C 180,E1 -20013.721,E2 -20013.721} C_VEL
LIN {X 0,Y 227.841,Z 496.071,A -85,B 0,C 180,E1 -20018.092,E2 -20018.092} C_VEL
LIN {X 0,Y 227.808,Z 496.09,A -85,B 0,C 180,E1 -20022.743,E2 -20022.743} C_VEL
LIN {X 0,Y 227.834,Z 496.091,A -85,B 0,C 180,E1 -20025.193,E2 -20025.193} C_VEL
LIN {X 0,Y 227.825,Z 496.093,A -85,B 0,C 180,E1 -20029.624,E2 -20029.624} C_VEL
LIN {X 0,Y 227.928,Z 496.217,A -85,B 0,C 180,E1 -20033.523,E2 -20033.523} C_VEL
LIN {X 0,Y 228.158,Z 497.196,A -85,B 0,C 180,E1 -20033.893,E2 -20033.893} C_VEL
LIN {X 0,Y 229.692,Z 499.931,A -85,B 0,C 180,E1 -20034.318,E2 -20034.318} C_VEL
LIN {X 0,Y 237.105,Z 512.386,A -85,B 0,C 180,E1 -20036.093,E2 -20036.093} C_VEL
LIN {X 0,Y 244.275,Z 525.691,A -85,B 0,C 180,E1 -20037.719,E2 -20037.719} C_VEL
LIN {X 0,Y 249.129,Z 535.995,A -85,B 0,C 180,E1 -20038.793,E2 -20038.793} C_VEL
LIN {X 0,Y 248.251,Z 574.114,A -85,B 0,C 180,E1 -20039.935,E2 -20039.935} C_VEL
LIN {X 0,Y 247.823,Z 587.2,A -85,B 0,C 180,E1 -20040.492,E2 -20040.492} C_VEL
LIN {X 0,Y 246.797,Z 600.632,A -85,B 0,C 180,E1 -20041.396,E2 -20041.396} C_VEL
LIN {X 0,Y 245.456,Z 612.911,A -85,B 0,C 180,E1 -20042.574,E2 -20042.574} C_VEL
LIN {X 0,Y 243.618,Z 624.386,A -85,B 0,C 180,E1 -20044.015,E2 -20044.015} C_VEL
LIN {X 0,Y 241.509,Z 635.121,A -85,B 0,C 180,E1 -20045.73,E2 -20045.73} C_VEL
LIN {X 0,Y 239.475,Z 644.311,A -85,B 0,C 180,E1 -20047.573,E2 -20047.573} C_VEL
LIN {X 0,Y 237.501,Z 652.659,A -85,B 0,C 180,E1 -20049.654,E2 -20049.654} C_VEL
LIN {X 0,Y 235.306,Z 660.767,A -85,B 0,C 180,E1 -20052.174,E2 -20052.174} C_VEL
LIN {X 0,Y 233.209,Z 667.872,A -85,B 0,C 180,E1 -20054.975,E2 -20054.975} C_VEL
LIN {X 0,Y 231.697,Z 673.24,A -85,B 0,C 180,E1 -20057.741,E2 -20057.741} C_VEL
LIN {X 0,Y 230.332,Z 677.128,A -85,B 0,C 180,E1 -20060.339,E2 -20060.339} C_VEL
LIN {X 0,Y 229.299,Z 679.997,A -85,B 0,C 180,E1 -20062.958,E2 -20062.958} C_VEL
LIN {X 0,Y 229.026,Z 681.337,A -85,B 0,C 180,E1 -20064.718,E2 -20064.718} C_VEL
LIN {X 0,Y 228.853,Z 682.286,A -85,B 0,C 180,E1 -20066.479,E2 -20066.479} C_VEL
LIN {X 0,Y 228.555,Z 683.114,A -85,B 0,C 180,E1 -20070,E2 -20070} C_VEL
LIN {X 0,Y 228.849,Z 682.344,A -85,B 0,C 180,E1 -20073.521,E2 -20073.521} C_VEL
LIN {X 0,Y 229.284,Z 680.114,A -85,B 0,C 180,E1 -20077.042,E2 -20077.042} C_VEL
LIN {X 0,Y 230.325,Z 677.287,A -85,B 0,C 180,E1 -20079.661,E2 -20079.661} C_VEL
LIN {X 0,Y 231.672,Z 673.456,A -85,B 0,C 180,E1 -20082.26,E2 -20082.26} C_VEL
LIN {X 0,Y 233.113,Z 668.372,A -85,B 0,C 180,E1 -20084.937,E2 -20084.937} C_VEL
LIN {X 0,Y 234.919,Z 662.335,A -85,B 0,C 180,E1 -20087.407,E2 -20087.407} C_VEL
LIN {X 0,Y 237.099,Z 654.548,A -85,B 0,C 180,E1 -20089.93,E2 -20089.93} C_VEL
LIN {X 0,Y 239.428,Z 644.87,A -85,B 0,C 180,E1 -20092.432,E2 -20092.432} C_VEL
LIN {X 0,Y 241.468,Z 635.814,A -85,B 0,C 180,E1 -20094.274,E2 -20094.274} C_VEL
LIN {X 0,Y 243.591,Z 625.293,A -85,B 0,C 180,E1 -20095.976,E2 -20095.976} C_VEL
LIN {X 0,Y 245.42,Z 613.759,A -85,B 0,C 180,E1 -20097.456,E2 -20097.456} C_VEL
LIN {X 0,Y 246.938,Z 602.455,A -85,B 0,C 180,E1 -20098.551,E2 -20098.551} C_VEL
LIN {X 0,Y 247.753,Z 590.081,A -85,B 0,C 180,E1 -20099.471,E2 -20099.471} C_VEL
LIN {X 0,Y 248.215,Z 576.743,A -85,B 0,C 180,E1 -20100.111,E2 -20100.111} C_VEL
LIN {X 0,Y 249.177,Z 535.928,A -85,B 0,C 180,E1 -20101.342,E2 -20101.342} C_VEL
LIN {X 0,Y 241.702,Z 520.652,A -85,B 0,C 180,E1 -20103.004,E2 -20103.004} C_VEL
LIN {X 0,Y 233.495,Z 506.27,A -85,B 0,C 180,E1 -20104.905,E2 -20104.905} C_VEL
LIN {X 0,Y 229.689,Z 499.958,A -85,B 0,C 180,E1 -20105.835,E2 -20105.835} C_VEL
LIN {X 0,Y 228.142,Z 497.182,A -85,B 0,C 180,E1 -20106.266,E2 -20106.266} C_VEL
LIN {X 0,Y 227.908,Z 496.16,A -85,B 0,C 180,E1 -20106.701,E2 -20106.701} C_VEL
LIN {X 0,Y 227.825,Z 496.097,A -85,B 0,C 180,E1 -20110.376,E2 -20110.376} C_VEL
LIN {X 0,Y 227.834,Z 496.098,A -85,B 0,C 180,E1 -20115.191,E2 -20115.191} C_VEL
LIN {X 0,Y 227.81,Z 496.06,A -85,B 0,C 180,E1 -20119.62,E2 -20119.62} C_VEL
LIN {X 0,Y 227.878,Z 496.1,A -85,B 0,C 180,E1 -20124.127,E2 -20124.127} C_VEL
LIN {X 0,Y 227.863,Z 496.04,A -85,B 0,C 180,E1 -20128.376,E2 -20128.376} C_VEL
LIN {X 0,Y 227.875,Z 496.074,A -85,B 0,C 180,E1 -20132.443,E2 -20132.443} C_VEL
LIN {X 0,Y 227.903,Z 496.084,A -85,B 0,C 180,E1 -20136.366,E2 -20136.366} C_VEL
LIN {X 0,Y 227.932,Z 496.092,A -85,B 0,C 180,E1 -20140.173,E2 -20140.173} C_VEL
LIN {X 0,Y 228.049,Z 496.057,A -85,B 0,C 180,E1 -20143.897,E2 -20143.897} C_VEL
LIN {X 0,Y 228.087,Z 496.073,A -85,B 0,C 180,E1 -20147.544,E2 -20147.544} C_VEL
LIN {X 0,Y 228.301,Z 496.023,A -85,B 0,C 180,E1 -20151.146,E2 -20151.146} C_VEL
LIN {X 0,Y 228.35,Z 496.034,A -85,B 0,C 180,E1 -20152.928,E2 -20152.928} C_VEL
LIN {X 0,Y 228.549,Z 495.993,A -85,B 0,C 180,E1 -20158.238,E2 -20158.238} C_VEL
LIN {X 0,Y 228.549,Z 496.008,A -85,B 0,C 180,E1 -20161.762,E2 -20161.762} C_VEL
LIN {X 0,Y 228.319,Z 496.041,A -85,B 0,C 180,E1 -20167.072,E2 -20167.072} C_VEL
LIN {X 0,Y 228.141,Z 496.044,A -85,B 0,C 180,E1 -20170.651,E2 -20170.651} C_VEL
LIN {X 0,Y 228.06,Z 496.077,A -85,B 0,C 180,E1 -20174.272,E2 -20174.272} C_VEL
LIN {X 0,Y 227.998,Z 496.044,A -85,B 0,C 180,E1 -20177.954,E2 -20177.954} C_VEL
LIN {X 0,Y 227.925,Z 496.091,A -85,B 0,C 180,E1 -20182.329,E2 -20182.329} C_VEL
LIN {X 0,Y 227.939,Z 496.06,A -85,B 0,C 180,E1 -20186.603,E2 -20186.603} C_VEL
LIN {X 0,Y 227.889,Z 496.096,A -85,B 0,C 180,E1 -20190.526,E2 -20190.526} C_VEL
LIN {X 0,Y 227.874,Z 496.078,A -85,B 0,C 180,E1 -20193.721,E2 -20193.721} C_VEL
LIN {X 0,Y 227.837,Z 496.088,A -85,B 0,C 180,E1 -20198.193,E2 -20198.193} C_VEL
LIN {X 0,Y 227.573,Z 496.409,A -85,B 0,C 180,E1 -20199.173,E2 -20199.173} C_VEL
LIN {X 0,Y 226.587,Z 497.85,A -85,B 0,C 180,E1 -20200.595,E2 -20200.595} C_VEL
LIN {X 0,Y 225.333,Z 500.11,A -85,B 0,C 180,E1 -20201.953,E2 -20201.953} C_VEL
LIN {X 0,Y 223.985,Z 503.957,A -85,B 0,C 180,E1 -20203.732,E2 -20203.732} C_VEL
LIN {X 0,Y 223.852,Z 507.084,A -85,B 0,C 180,E1 -20205.051,E2 -20205.051} C_VEL
LIN {X 0,Y 224.075,Z 508.118,A -85,B 0,C 180,E1 -20205.488,E2 -20205.488} C_VEL
LIN {X 0,Y 226.292,Z 516.514,A -85,B 0,C 180,E1 -20208.893,E2 -20208.893} C_VEL
LIN {X 0,Y 228.914,Z 528.027,A -85,B 0,C 180,E1 -20213.116,E2 -20213.116} C_VEL
LIN {X 0,Y 233.605,Z 539.657,A -85,B 0,C 180,E1 -20214.414,E2 -20214.414} C_VEL
LIN {X 0,Y 237.133,Z 568.614,A -85,B 0,C 180,E1 -20216.03,E2 -20216.03} C_VEL
LIN {X 0,Y 239.789,Z 599.668,A -85,B 0,C 180,E1 -20217.516,E2 -20217.516} C_VEL
LIN {X 0,Y 240.521,Z 611.314,A -85,B 0,C 180,E1 -20218.021,E2 -20218.021} C_VEL
LIN {X 0,Y 239.155,Z 641.206,A -85,B 0,C 180,E1 -20218.918,E2 -20218.918} C_VEL
LIN {X 0,Y 237.909,Z 654.717,A -85,B 0,C 180,E1 -20219.65,E2 -20219.65} C_VEL
LIN {X 0,Y 236.373,Z 665.621,A -85,B 0,C 180,E1 -20220.499,E2 -20220.499} C_VEL
LIN {X 0,Y 234.027,Z 677.899,A -85,B 0,C 180,E1 -20221.773,E2 -20221.773} C_VEL
LIN {X 0,Y 231.363,Z 689.549,A -85,B 0,C 180,E1 -20223.382,E2 -20223.382} C_VEL
LIN {X 0,Y 228.937,Z 698.985,A -85,B 0,C 180,E1 -20225.033,E2 -20225.033} C_VEL
LIN {X 0,Y 226.361,Z 708.712,A -85,B 0,C 180,E1 -20227.164,E2 -20227.164} C_VEL
LIN {X 0,Y 224.213,Z 716.726,A -85,B 0,C 180,E1 -20229.352,E2 -20229.352} C_VEL
LIN {X 0,Y 222.367,Z 723.394,A -85,B 0,C 180,E1 -20231.576,E2 -20231.576} C_VEL
LIN {X 0,Y 220.895,Z 730.036,A -85,B 0,C 180,E1 -20234.31,E2 -20234.31} C_VEL
LIN {X 0,Y 219.937,Z 735.356,A -85,B 0,C 180,E1 -20237.075,E2 -20237.075} C_VEL
LIN {X 0,Y 219.543,Z 739.545,A -85,B 0,C 180,E1 -20239.86,E2 -20239.86} C_VEL
LIN {X 0,Y 219.675,Z 742.702,A -85,B 0,C 180,E1 -20242.648,E2 -20242.648} C_VEL
LIN {X 0,Y 219.88,Z 744.226,A -85,B 0,C 180,E1 -20244.498,E2 -20244.498} C_VEL
LIN {X 0,Y 220.244,Z 745.343,A -85,B 0,C 180,E1 -20246.341,E2 -20246.341} C_VEL
LIN {X 0,Y 221.069,Z 746.333,A -85,B 0,C 180,E1 -20250,E2 -20250} C_VEL
LIN {X 0,Y 220.259,Z 745.329,A -85,B 0,C 180,E1 -20253.659,E2 -20253.659} C_VEL
LIN {X 0,Y 219.925,Z 744.21,A -85,B 0,C 180,E1 -20255.501,E2 -20255.501} C_VEL
LIN {X 0,Y 219.577,Z 741.699,A -85,B 0,C 180,E1 -20258.281,E2 -20258.281} C_VEL
LIN {X 0,Y 219.632,Z 738.191,A -85,B 0,C 180,E1 -20261.069,E2 -20261.069} C_VEL
LIN {X 0,Y 220.237,Z 733.622,A -85,B 0,C 180,E1 -20263.847,E2 -20263.847} C_VEL
LIN {X 0,Y 221.376,Z 727.869,A -85,B 0,C 180,E1 -20266.602,E2 -20266.602} C_VEL
LIN {X 0,Y 222.792,Z 722.061,A -85,B 0,C 180,E1 -20268.852,E2 -20268.852} C_VEL
LIN {X 0,Y 225.016,Z 713.546,A -85,B 0,C 180,E1 -20271.53,E2 -20271.53} C_VEL
LIN {X 0,Y 227.372,Z 704.898,A -85,B 0,C 180,E1 -20273.692,E2 -20273.692} C_VEL
LIN {X 0,Y 230.109,Z 694.26,A -85,B 0,C 180,E1 -20275.799,E2 -20275.799} C_VEL
LIN {X 0,Y 233.047,Z 682.347,A -85,B 0,C 180,E1 -20277.623,E2 -20277.623} C_VEL
LIN {X 0,Y 235.448,Z 670.347,A -85,B 0,C 180,E1 -20279.015,E2 -20279.015} C_VEL
LIN {X 0,Y 237.345,Z 657.865,A -85,B 0,C 180,E1 -20280.101,E2 -20280.101} C_VEL
LIN {X 0,Y 238.867,Z 644.807,A -85,B 0,C 180,E1 -20280.879,E2 -20280.879} C_VEL
LIN {X 0,Y 239.628,Z 630.992,A -85,B 0,C 180,E1 -20281.385,E2 -20281.385} C_VEL
LIN {X 0,Y 240.363,Z 609.532,A -85,B 0,C 180,E1 -20282.012,E2 -20282.012} C_VEL
LIN {X 0,Y 237.86,Z 576.941,A -85,B 0,C 180,E1 -20283.511,E2 -20283.511} C_VEL
LIN {X 0,Y 234.576,Z 547.438,A -85,B 0,C 180,E1 -20285.085,E2 -20285.085} C_VEL
LIN {X 0,Y 233.373,Z 538.818,A -85,B 0,C 180,E1 -20285.6,E2 -20285.6} C_VEL
LIN {X 0,Y 228.835,Z 527.901,A -85,B 0,C 180,E1 -20286.858,E2 -20286.858} C_VEL
LIN {X 0,Y 226.524,Z 517.519,A -85,B 0,C 180,E1 -20290.656,E2 -20290.656} C_VEL
LIN {X 0,Y 224.082,Z 508.037,A -85,B 0,C 180,E1 -20294.478,E2 -20294.478} C_VEL
LIN {X 0,Y 221.539,Z 499.554,A -85,B 0,C 180,E1 -20298.226,E2 -20298.226} C_VEL
LIN {X 0,Y 220.81,Z 497.036,A -85,B 0,C 180,E1 -20299.496,E2 -20299.496} C_VEL
LIN {X 0,Y 220.822,Z 496.966,A -85,B 0,C 180,E1 -20302.792,E2 -20302.792} C_VEL
LIN {X 0,Y 220.814,Z 496.957,A -85,B 0,C 180,E1 -20307.243,E2 -20307.243} C_VEL
LIN {X 0,Y 220.833,Z 496.955,A -85,B 0,C 180,E1 -20311.486,E2 -20311.486} C_VEL
LIN {X 0,Y 220.863,Z 496.965,A -85,B 0,C 180,E1 -20315.565,E2 -20315.565} C_VEL
LIN {X 0,Y 220.887,Z 496.935,A -85,B 0,C 180,E1 -20319.513,E2 -20319.513} C_VEL
LIN {X 0,Y 221.012,Z 496.932,A -85,B 0,C 180,E1 -20323.37,E2 -20323.37} C_VEL
LIN {X 0,Y 221.007,Z 496.946,A -85,B 0,C 180,E1 -20327.138,E2 -20327.138} C_VEL
LIN {X 0,Y 221.2,Z 496.923,A -85,B 0,C 180,E1 -20330.859,E2 -20330.859} C_VEL
LIN {X 0,Y 221.255,Z 496.924,A -85,B 0,C 180,E1 -20332.7,E2 -20332.7} C_VEL
LIN {X 0,Y 221.507,Z 496.889,A -85,B 0,C 180,E1 -20338.182,E2 -20338.182} C_VEL
LIN {X 0,Y 221.508,Z 496.872,A -85,B 0,C 180,E1 -20341.818,E2 -20341.818} C_VEL
LIN {X 0,Y 221.255,Z 496.918,A -85,B 0,C 180,E1 -20347.3,E2 -20347.3} C_VEL
LIN {X 0,Y 221.062,Z 496.933,A -85,B 0,C 180,E1 -20350.997,E2 -20350.997} C_VEL
LIN {X 0,Y 221.01,Z 496.934,A -85,B 0,C 180,E1 -20356.63,E2 -20356.63} C_VEL
LIN {X 0,Y 220.88,Z 496.965,A -85,B 0,C 180,E1 -20360.488,E2 -20360.488} C_VEL
LIN {X 0,Y 220.858,Z 496.97,A -85,B 0,C 180,E1 -20364.436,E2 -20364.436} C_VEL
LIN {X 0,Y 220.823,Z 496.931,A -85,B 0,C 180,E1 -20368.516,E2 -20368.516} C_VEL
LIN {X 0,Y 220.813,Z 496.929,A -85,B 0,C 180,E1 -20372.757,E2 -20372.757} C_VEL
LIN {X 0,Y 220.807,Z 496.962,A -85,B 0,C 180,E1 -20377.279,E2 -20377.279} C_VEL
LIN {X 0,Y 220.764,Z 496.951,A -85,B 0,C 180,E1 -20381.954,E2 -20381.954} C_VEL
LIN {X 0,Y 220.774,Z 496.963,A -85,B 0,C 180,E1 -20385.547,E2 -20385.547} C_VEL
LIN {X 0,Y 220.806,Z 496.983,A -85,B 0,C 180,E1 -20390.464,E2 -20390.464} C_VEL
LIN {X 0,Y 220.833,Z 497.184,A -85,B 0,C 180,E1 -20392.177,E2 -20392.177} C_VEL
LIN {X 0,Y 221.096,Z 498.209,A -85,B 0,C 180,E1 -20392.543,E2 -20392.543} C_VEL
LIN {X 0,Y 222.721,Z 500.975,A -85,B 0,C 180,E1 -20393.011,E2 -20393.011} C_VEL
LIN {X 0,Y 223.963,Z 502.909,A -85,B 0,C 180,E1 -20393.336,E2 -20393.336} C_VEL
LIN {X 0,Y 230.327,Z 513.383,A -85,B 0,C 180,E1 -20394.945,E2 -20394.945} C_VEL
LIN {X 0,Y 237.667,Z 526.74,A -85,B 0,C 180,E1 -20396.704,E2 -20396.704} C_VEL
LIN {X 0,Y 243.117,Z 538.092,A -85,B 0,C 180,E1 -20397.968,E2 -20397.968} C_VEL
LIN {X 0,Y 242.182,Z 574.577,A -85,B 0,C 180,E1 -20399.082,E2 -20399.082} C_VEL
LIN {X 0,Y 241.738,Z 588.049,A -85,B 0,C 180,E1 -20399.662,E2 -20399.662} C_VEL
LIN {X 0,Y 240.651,Z 601.629,A -85,B 0,C 180,E1 -20400.595,E2 -20400.595} C_VEL
LIN {X 0,Y 239.24,Z 613.905,A -85,B 0,C 180,E1 -20401.799,E2 -20401.799} C_VEL
LIN {X 0,Y 237.325,Z 625.377,A -85,B 0,C 180,E1 -20403.272,E2 -20403.272} C_VEL
LIN {X 0,Y 235.12,Z 636.113,A -85,B 0,C 180,E1 -20405.026,E2 -20405.026} C_VEL
LIN {X 0,Y 232.993,Z 645.302,A -85,B 0,C 180,E1 -20406.913,E2 -20406.913} C_VEL
LIN {X 0,Y 230.924,Z 653.649,A -85,B 0,C 180,E1 -20409.048,E2 -20409.048} C_VEL
LIN {X 0,Y 228.625,Z 661.757,A -85,B 0,C 180,E1 -20411.634,E2 -20411.634} C_VEL
LIN {X 0,Y 226.429,Z 668.862,A -85,B 0,C 180,E1 -20414.514,E2 -20414.514} C_VEL
LIN {X 0,Y 224.834,Z 674.23,A -85,B 0,C 180,E1 -20417.361,E2 -20417.361} C_VEL
LIN {X 0,Y 223.407,Z 678.117,A -85,B 0,C 180,E1 -20420.037,E2 -20420.037} C_VEL
LIN {X 0,Y 222.323,Z 680.987,A -85,B 0,C 180,E1 -20422.736,E2 -20422.736} C_VEL
LIN {X 0,Y 222.028,Z 682.326,A -85,B 0,C 180,E1 -20424.551,E2 -20424.551} C_VEL
LIN {X 0,Y 221.841,Z 683.275,A -85,B 0,C 180,E1 -20426.367,E2 -20426.367} C_VEL
LIN {X 0,Y 221.527,Z 684.102,A -85,B 0,C 180,E1 -20430,E2 -20430} C_VEL
LIN {X 0,Y 221.837,Z 683.331,A -85,B 0,C 180,E1 -20433.633,E2 -20433.633} C_VEL
LIN {X 0,Y 222.308,Z 681.102,A -85,B 0,C 180,E1 -20437.265,E2 -20437.265} C_VEL
LIN {X 0,Y 223.4,Z 678.275,A -85,B 0,C 180,E1 -20439.964,E2 -20439.964} C_VEL
LIN {X 0,Y 224.809,Z 674.443,A -85,B 0,C 180,E1 -20442.64,E2 -20442.64} C_VEL
LIN {X 0,Y 226.33,Z 669.359,A -85,B 0,C 180,E1 -20445.395,E2 -20445.395} C_VEL
LIN {X 0,Y 228.223,Z 663.321,A -85,B 0,C 180,E1 -20447.935,E2 -20447.935} C_VEL
LIN {X 0,Y 230.504,Z 655.534,A -85,B 0,C 180,E1 -20450.525,E2 -20450.525} C_VEL
LIN {X 0,Y 232.946,Z 645.856,A -85,B 0,C 180,E1 -20453.092,E2 -20453.092} C_VEL
LIN {X 0,Y 235.066,Z 636.8,A -85,B 0,C 180,E1 -20454.98,E2 -20454.98} C_VEL
LIN {X 0,Y 237.293,Z 626.276,A -85,B 0,C 180,E1 -20456.719,E2 -20456.719} C_VEL
LIN {X 0,Y 239.204,Z 614.741,A -85,B 0,C 180,E1 -20458.233,E2 -20458.233} C_VEL
LIN {X 0,Y 240.786,Z 603.436,A -85,B 0,C 180,E1 -20459.351,E2 -20459.351} C_VEL
LIN {X 0,Y 241.67,Z 590.79,A -85,B 0,C 180,E1 -20460.307,E2 -20460.307} C_VEL
LIN {X 0,Y 242.158,Z 577.594,A -85,B 0,C 180,E1 -20460.95,E2 -20460.95} C_VEL
LIN {X 0,Y 243.129,Z 537.999,A -85,B 0,C 180,E1 -20462.176,E2 -20462.176} C_VEL
LIN {X 0,Y 235.595,Z 522.736,A -85,B 0,C 180,E1 -20463.935,E2 -20463.935} C_VEL
LIN {X 0,Y 227.044,Z 507.825,A -85,B 0,C 180,E1 -20466.031,E2 -20466.031} C_VEL
LIN {X 0,Y 222.83,Z 501.107,A -85,B 0,C 180,E1 -20467.12,E2 -20467.12} C_VEL
LIN {X 0,Y 221.202,Z 498.56,A -85,B 0,C 180,E1 -20467.568,E2 -20467.568} C_VEL
LIN {X 0,Y 220.849,Z 497.308,A -85,B 0,C 180,E1 -20467.88,E2 -20467.88} C_VEL
LIN {X 0,Y 220.795,Z 496.978,A -85,B 0,C 180,E1 -20468.367,E2 -20468.367} C_VEL
LIN {X 0,Y 220.766,Z 496.952,A -85,B 0,C 180,E1 -20472.929,E2 -20472.929} C_VEL
LIN {X 0,Y 220.764,Z 496.974,A -85,B 0,C 180,E1 -20477.07,E2 -20477.07} C_VEL
LIN {X 0,Y 220.784,Z 496.934,A -85,B 0,C 180,E1 -20480.458,E2 -20480.458} C_VEL
LIN {X 0,Y 220.822,Z 496.96,A -85,B 0,C 180,E1 -20482.792,E2 -20482.792} C_VEL
LIN {X 0,Y 220.813,Z 496.931,A -85,B 0,C 180,E1 -20487.243,E2 -20487.243} C_VEL
LIN {X 0,Y 220.823,Z 496.931,A -85,B 0,C 180,E1 -20491.484,E2 -20491.484} C_VEL
LIN {X 0,Y 220.858,Z 496.97,A -85,B 0,C 180,E1 -20495.564,E2 -20495.564} C_VEL
LIN {X 0,Y 220.88,Z 496.964,A -85,B 0,C 180,E1 -20499.512,E2 -20499.512} C_VEL
LIN {X 0,Y 221.01,Z 496.934,A -85,B 0,C 180,E1 -20503.37,E2 -20503.37} C_VEL
LIN {X 0,Y 221.107,Z 496.927,A -85,B 0,C 180,E1 -20509.005,E2 -20509.005} C_VEL
LIN {X 0,Y 221.301,Z 496.911,A -85,B 0,C 180,E1 -20512.702,E2 -20512.702} C_VEL
LIN {X 0,Y 221.507,Z 496.869,A -85,B 0,C 180,E1 -20518.182,E2 -20518.182} C_VEL
LIN {X 0,Y 221.507,Z 496.885,A -85,B 0,C 180,E1 -20521.818,E2 -20521.818} C_VEL
LIN {X 0,Y 221.255,Z 496.923,A -85,B 0,C 180,E1 -20527.3,E2 -20527.3} C_VEL
LIN {X 0,Y 221.063,Z 496.925,A -85,B 0,C 180,E1 -20530.997,E2 -20530.997} C_VEL
LIN {X 0,Y 220.992,Z 496.957,A -85,B 0,C 180,E1 -20534.739,E2 -20534.739} C_VEL
LIN {X 0,Y 220.917,Z 496.922,A -85,B 0,C 180,E1 -20538.55,E2 -20538.55} C_VEL
LIN {X 0,Y 220.892,Z 496.97,A -85,B 0,C 180,E1 -20542.682,E2 -20542.682} C_VEL
LIN {X 0,Y 220.882,Z 496.938,A -85,B 0,C 180,E1 -20547.016,E2 -20547.016} C_VEL
LIN {X 0,Y 220.86,Z 496.972,A -85,B 0,C 180,E1 -20550.779,E2 -20550.779} C_VEL
LIN {X 0,Y 220.799,Z 496.971,A -85,B 0,C 180,E1 -20554.955,E2 -20554.955} C_VEL
LIN {X 0,Y 220.804,Z 496.972,A -85,B 0,C 180,E1 -20559.538,E2 -20559.538} C_VEL
LIN {X 0,Y 220.843,Z 497.249,A -85,B 0,C 180,E1 -20560.615,E2 -20560.615} C_VEL
LIN {X 0,Y 223.361,Z 505.661,A -85,B 0,C 180,E1 -20564.434,E2 -20564.434} C_VEL
LIN {X 0,Y 224.075,Z 508.118,A -85,B 0,C 180,E1 -20565.488,E2 -20565.488} C_VEL
LIN {X 0,Y 224.026,Z 510.391,A -85,B 0,C 180,E1 -20566.316,E2 -20566.316} C_VEL
LIN {X 0,Y 222.237,Z 514.663,A -85,B 0,C 180,E1 -20567.566,E2 -20567.566} C_VEL
LIN {X 0,Y 220.364,Z 519.001,A -85,B 0,C 180,E1 -20568.83,E2 -20568.83} C_VEL
LIN {X 0,Y 220.225,Z 521.387,A -85,B 0,C 180,E1 -20569.669,E2 -20569.669} C_VEL
LIN {X 0,Y 221.391,Z 526.598,A -85,B 0,C 180,E1 -20571.621,E2 -20571.621} C_VEL
LIN {X 0,Y 225.936,Z 537.122,A -85,B 0,C 180,E1 -20572.962,E2 -20572.962} C_VEL
LIN {X 0,Y 228.058,Z 542.453,A -85,B 0,C 180,E1 -20573.552,E2 -20573.552} C_VEL
LIN {X 0,Y 231.503,Z 572.545,A -85,B 0,C 180,E1 -20575.264,E2 -20575.264} C_VEL
LIN {X 0,Y 234.235,Z 606.79,A -85,B 0,C 180,E1 -20576.932,E2 -20576.932} C_VEL
LIN {X 0,Y 234.329,Z 614.176,A -85,B 0,C 180,E1 -20577.208,E2 -20577.208} C_VEL
LIN {X 0,Y 233.078,Z 640.521,A -85,B 0,C 180,E1 -20578.03,E2 -20578.03} C_VEL
LIN {X 0,Y 231.775,Z 653.853,A -85,B 0,C 180,E1 -20578.768,E2 -20578.768} C_VEL
LIN {X 0,Y 230.021,Z 665.745,A -85,B 0,C 180,E1 -20579.727,E2 -20579.727} C_VEL
LIN {X 0,Y 227.783,Z 676.903,A -85,B 0,C 180,E1 -20580.926,E2 -20580.926} C_VEL
LIN {X 0,Y 225.022,Z 688.552,A -85,B 0,C 180,E1 -20582.57,E2 -20582.57} C_VEL
LIN {X 0,Y 222.204,Z 699.069,A -85,B 0,C 180,E1 -20584.474,E2 -20584.474} C_VEL
LIN {X 0,Y 219.79,Z 707.709,A -85,B 0,C 180,E1 -20586.441,E2 -20586.441} C_VEL
LIN {X 0,Y 217.53,Z 715.722,A -85,B 0,C 180,E1 -20588.687,E2 -20588.687} C_VEL
LIN {X 0,Y 215.654,Z 722.4,A -85,B 0,C 180,E1 -20590.981,E2 -20590.981} C_VEL
LIN {X 0,Y 214.213,Z 727.995,A -85,B 0,C 180,E1 -20593.318,E2 -20593.318} C_VEL
LIN {X 0,Y 212.959,Z 734.35,A -85,B 0,C 180,E1 -20596.644,E2 -20596.644} C_VEL
LIN {X 0,Y 212.504,Z 738.54,A -85,B 0,C 180,E1 -20599.52,E2 -20599.52} C_VEL
LIN {X 0,Y 212.612,Z 741.868,A -85,B 0,C 180,E1 -20602.598,E2 -20602.598} C_VEL
LIN {X 0,Y 213.176,Z 744.348,A -85,B 0,C 180,E1 -20606.219,E2 -20606.219} C_VEL
LIN {X 0,Y 214.025,Z 745.343,A -85,B 0,C 180,E1 -20610,E2 -20610} C_VEL
LIN {X 0,Y 213.194,Z 744.333,A -85,B 0,C 180,E1 -20613.78,E2 -20613.78} C_VEL
LIN {X 0,Y 212.615,Z 741.833,A -85,B 0,C 180,E1 -20617.408,E2 -20617.408} C_VEL
LIN {X 0,Y 212.508,Z 738.49,A -85,B 0,C 180,E1 -20620.48,E2 -20620.48} C_VEL
LIN {X 0,Y 212.964,Z 734.28,A -85,B 0,C 180,E1 -20623.356,E2 -20623.356} C_VEL
LIN {X 0,Y 214.251,Z 727.902,A -85,B 0,C 180,E1 -20626.679,E2 -20626.679} C_VEL
LIN {X 0,Y 215.847,Z 721.717,A -85,B 0,C 180,E1 -20629.223,E2 -20629.223} C_VEL
LIN {X 0,Y 217.95,Z 714.058,A -85,B 0,C 180,E1 -20631.766,E2 -20631.766} C_VEL
LIN {X 0,Y 220.33,Z 705.725,A -85,B 0,C 180,E1 -20633.997,E2 -20633.997} C_VEL
LIN {X 0,Y 223.077,Z 695.6,A -85,B 0,C 180,E1 -20636.171,E2 -20636.171} C_VEL
LIN {X 0,Y 226.055,Z 684.217,A -85,B 0,C 180,E1 -20638.049,E2 -20638.049} C_VEL
LIN {X 0,Y 228.551,Z 673.086,A -85,B 0,C 180,E1 -20639.472,E2 -20639.472} C_VEL
LIN {X 0,Y 230.472,Z 661.865,A -85,B 0,C 180,E1 -20640.588,E2 -20640.588} C_VEL
LIN {X 0,Y 232.25,Z 649.025,A -85,B 0,C 180,E1 -20641.501,E2 -20641.501} C_VEL
LIN {X 0,Y 233.334,Z 635.272,A -85,B 0,C 180,E1 -20642.129,E2 -20642.129} C_VEL
LIN {X 0,Y 234.308,Z 610.4,A -85,B 0,C 180,E1 -20642.875,E2 -20642.875} C_VEL
LIN {X 0,Y 231.985,Z 578.799,A -85,B 0,C 180,E1 -20644.372,E2 -20644.372} C_VEL
LIN {X 0,Y 228.859,Z 549.488,A -85,B 0,C 180,E1 -20645.981,E2 -20645.981} C_VEL
LIN {X 0,Y 227.656,Z 541.301,A -85,B 0,C 180,E1 -20646.503,E2 -20646.503} C_VEL
LIN {X 0,Y 222.844,Z 530.246,A -85,B 0,C 180,E1 -20647.825,E2 -20647.825} C_VEL
LIN {X 0,Y 221.331,Z 526.433,A -85,B 0,C 180,E1 -20648.366,E2 -20648.366} C_VEL
LIN {X 0,Y 219.317,Z 517.467,A -85,B 0,C 180,E1 -20651.838,E2 -20651.838} C_VEL
LIN {X 0,Y 216.713,Z 507.727,A -85,B 0,C 180,E1 -20656.006,E2 -20656.006} C_VEL
LIN {X 0,Y 213.783,Z 497.985,A -85,B 0,C 180,E1 -20660.664,E2 -20660.664} C_VEL
LIN {X 0,Y 213.769,Z 497.842,A -85,B 0,C 180,E1 -20665.275,E2 -20665.275} C_VEL
LIN {X 0,Y 213.792,Z 497.846,A -85,B 0,C 180,E1 -20668.724,E2 -20668.724} C_VEL
LIN {X 0,Y 213.823,Z 497.818,A -85,B 0,C 180,E1 -20672.603,E2 -20672.603} C_VEL
LIN {X 0,Y 213.848,Z 497.847,A -85,B 0,C 180,E1 -20676.953,E2 -20676.953} C_VEL
LIN {X 0,Y 213.939,Z 497.802,A -85,B 0,C 180,E1 -20682.803,E2 -20682.803} C_VEL
LIN {X 0,Y 213.948,Z 497.829,A -85,B 0,C 180,E1 -20686.706,E2 -20686.706} C_VEL
LIN {X 0,Y 214.137,Z 497.799,A -85,B 0,C 180,E1 -20690.555,E2 -20690.555} C_VEL
LIN {X 0,Y 214.096,Z 497.798,A -85,B 0,C 180,E1 -20694.348,E2 -20694.348} C_VEL
LIN {X 0,Y 214.441,Z 497.769,A -85,B 0,C 180,E1 -20698.122,E2 -20698.122} C_VEL
LIN {X 0,Y 214.549,Z 497.757,A -85,B 0,C 180,E1 -20700,E2 -20700} C_VEL
LIN {X 0,Y 214.441,Z 497.751,A -85,B 0,C 180,E1 -20701.878,E2 -20701.878} C_VEL
LIN {X 0,Y 214.194,Z 497.793,A -85,B 0,C 180,E1 -20707.542,E2 -20707.542} C_VEL
LIN {X 0,Y 213.994,Z 497.817,A -85,B 0,C 180,E1 -20711.365,E2 -20711.365} C_VEL
LIN {X 0,Y 213.924,Z 497.818,A -85,B 0,C 180,E1 -20715.238,E2 -20715.238} C_VEL
LIN {X 0,Y 213.832,Z 497.85,A -85,B 0,C 180,E1 -20719.188,E2 -20719.188} C_VEL
LIN {X 0,Y 213.807,Z 497.835,A -85,B 0,C 180,E1 -20723.232,E2 -20723.232} C_VEL
LIN {X 0,Y 213.826,Z 497.824,A -85,B 0,C 180,E1 -20727.451,E2 -20727.451} C_VEL
LIN {X 0,Y 213.765,Z 497.793,A -85,B 0,C 180,E1 -20731.738,E2 -20731.738} C_VEL
LIN {X 0,Y 213.741,Z 497.859,A -85,B 0,C 180,E1 -20736.289,E2 -20736.289} C_VEL
LIN {X 0,Y 213.704,Z 497.819,A -85,B 0,C 180,E1 -20741.127,E2 -20741.127} C_VEL
LIN {X 0,Y 213.706,Z 497.864,A -85,B 0,C 180,E1 -20743.679,E2 -20743.679} C_VEL
LIN {X 0,Y 213.705,Z 497.833,A -85,B 0,C 180,E1 -20746.345,E2 -20746.345} C_VEL
LIN {X 0,Y 213.794,Z 498.021,A -85,B 0,C 180,E1 -20750.686,E2 -20750.686} C_VEL
LIN {X 0,Y 214.057,Z 499.2,A -85,B 0,C 180,E1 -20751.081,E2 -20751.081} C_VEL
LIN {X 0,Y 215.619,Z 501.781,A -85,B 0,C 180,E1 -20751.555,E2 -20751.555} C_VEL
LIN {X 0,Y 216.7,Z 503.345,A -85,B 0,C 180,E1 -20751.856,E2 -20751.856} C_VEL
LIN {X 0,Y 224.223,Z 515.452,A -85,B 0,C 180,E1 -20753.882,E2 -20753.882} C_VEL
LIN {X 0,Y 231.981,Z 529.678,A -85,B 0,C 180,E1 -20755.849,E2 -20755.849} C_VEL
LIN {X 0,Y 237.053,Z 540.092,A -85,B 0,C 180,E1 -20757.081,E2 -20757.081} C_VEL
LIN {X 0,Y 236.012,Z 581.954,A -85,B 0,C 180,E1 -20758.439,E2 -20758.439} C_VEL
LIN {X 0,Y 235.279,Z 595.294,A -85,B 0,C 180,E1 -20759.196,E2 -20759.196} C_VEL
LIN {X 0,Y 234.084,Z 607.267,A -85,B 0,C 180,E1 -20760.183,E2 -20760.183} C_VEL
LIN {X 0,Y 232.361,Z 619.545,A -85,B 0,C 180,E1 -20761.548,E2 -20761.548} C_VEL
LIN {X 0,Y 230.065,Z 631.094,A -85,B 0,C 180,E1 -20763.22,E2 -20763.22} C_VEL
LIN {X 0,Y 227.745,Z 641.409,A -85,B 0,C 180,E1 -20765.137,E2 -20765.137} C_VEL
LIN {X 0,Y 225.627,Z 649.819,A -85,B 0,C 180,E1 -20767.086,E2 -20767.086} C_VEL
LIN {X 0,Y 223.544,Z 657.545,A -85,B 0,C 180,E1 -20769.287,E2 -20769.287} C_VEL
LIN {X 0,Y 221.178,Z 665.212,A -85,B 0,C 180,E1 -20772.001,E2 -20772.001} C_VEL
LIN {X 0,Y 219.333,Z 670.956,A -85,B 0,C 180,E1 -20774.574,E2 -20774.574} C_VEL
LIN {X 0,Y 217.982,Z 675.219,A -85,B 0,C 180,E1 -20776.957,E2 -20776.957} C_VEL
LIN {X 0,Y 216.489,Z 679.107,A -85,B 0,C 180,E1 -20779.715,E2 -20779.715} C_VEL
LIN {X 0,Y 215.351,Z 681.976,A -85,B 0,C 180,E1 -20782.499,E2 -20782.499} C_VEL
LIN {X 0,Y 215.031,Z 683.315,A -85,B 0,C 180,E1 -20784.373,E2 -20784.373} C_VEL
LIN {X 0,Y 214.829,Z 684.263,A -85,B 0,C 180,E1 -20786.249,E2 -20786.249} C_VEL
LIN {X 0,Y 214.5,Z 685.09,A -85,B 0,C 180,E1 -20790,E2 -20790} C_VEL
LIN {X 0,Y 214.825,Z 684.319,A -85,B 0,C 180,E1 -20793.751,E2 -20793.751} C_VEL
LIN {X 0,Y 215.335,Z 682.09,A -85,B 0,C 180,E1 -20797.501,E2 -20797.501} C_VEL
LIN {X 0,Y 216.481,Z 679.262,A -85,B 0,C 180,E1 -20800.285,E2 -20800.285} C_VEL
LIN {X 0,Y 217.957,Z 675.43,A -85,B 0,C 180,E1 -20803.045,E2 -20803.045} C_VEL
LIN {X 0,Y 219.562,Z 670.345,A -85,B 0,C 180,E1 -20805.882,E2 -20805.882} C_VEL
LIN {X 0,Y 221.547,Z 664.308,A -85,B 0,C 180,E1 -20808.495,E2 -20808.495} C_VEL
LIN {X 0,Y 223.935,Z 656.52,A -85,B 0,C 180,E1 -20811.156,E2 -20811.156} C_VEL
LIN {X 0,Y 226.497,Z 646.841,A -85,B 0,C 180,E1 -20813.789,E2 -20813.789} C_VEL
LIN {X 0,Y 228.693,Z 637.788,A -85,B 0,C 180,E1 -20815.726,E2 -20815.726} C_VEL
LIN {X 0,Y 231.029,Z 627.262,A -85,B 0,C 180,E1 -20817.504,E2 -20817.504} C_VEL
LIN {X 0,Y 233.071,Z 615.567,A -85,B 0,C 180,E1 -20819.067,E2 -20819.067} C_VEL
LIN {X 0,Y 234.727,Z 604.073,A -85,B 0,C 180,E1 -20820.223,E2 -20820.223} C_VEL
LIN {X 0,Y 235.653,Z 591.534,A -85,B 0,C 180,E1 -20821.182,E2 -20821.182} C_VEL
LIN {X 0,Y 236.154,Z 578.562,A -85,B 0,C 180,E1 -20821.828,E2 -20821.828} C_VEL
LIN {X 0,Y 237.119,Z 540.122,A -85,B 0,C 180,E1 -20823.054,E2 -20823.054} C_VEL
LIN {X 0,Y 230.158,Z 526,A -85,B 0,C 180,E1 -20824.761,E2 -20824.761} C_VEL
LIN {X 0,Y 221.731,Z 511.278,A -85,B 0,C 180,E1 -20826.933,E2 -20826.933} C_VEL
LIN {X 0,Y 217.918,Z 505.412,A -85,B 0,C 180,E1 -20827.961,E2 -20827.961} C_VEL
LIN {X 0,Y 215.922,Z 502.11,A -85,B 0,C 180,E1 -20828.529,E2 -20828.529} C_VEL
LIN {X 0,Y 214.289,Z 499.785,A -85,B 0,C 180,E1 -20828.996,E2 -20828.996} C_VEL
LIN {X 0,Y 213.847,Z 498.337,A -85,B 0,C 180,E1 -20829.308,E2 -20829.308} C_VEL
LIN {X 0,Y 213.776,Z 497.882,A -85,B 0,C 180,E1 -20829.872,E2 -20829.872} C_VEL
LIN {X 0,Y 213.705,Z 497.834,A -85,B 0,C 180,E1 -20833.677,E2 -20833.677} C_VEL
LIN {X 0,Y 213.706,Z 497.867,A -85,B 0,C 180,E1 -20836.343,E2 -20836.343} C_VEL
LIN {X 0,Y 213.708,Z 497.818,A -85,B 0,C 180,E1 -20839.144,E2 -20839.144} C_VEL
LIN {X 0,Y 213.741,Z 497.858,A -85,B 0,C 180,E1 -20843.711,E2 -20843.711} C_VEL
LIN {X 0,Y 213.777,Z 497.789,A -85,B 0,C 180,E1 -20848.731,E2 -20848.731} C_VEL
LIN {X 0,Y 213.823,Z 497.825,A -85,B 0,C 180,E1 -20852.603,E2 -20852.603} C_VEL
LIN {X 0,Y 213.815,Z 497.833,A -85,B 0,C 180,E1 -20856.973,E2 -20856.973} C_VEL
LIN {X 0,Y 213.939,Z 497.818,A -85,B 0,C 180,E1 -20862.803,E2 -20862.803} C_VEL
LIN {X 0,Y 213.973,Z 497.831,A -85,B 0,C 180,E1 -20866.708,E2 -20866.708} C_VEL
LIN {X 0,Y 214.163,Z 497.782,A -85,B 0,C 180,E1 -20870.556,E2 -20870.556} C_VEL
LIN {X 0,Y 214.236,Z 497.787,A -85,B 0,C 180,E1 -20872.46,E2 -20872.46} C_VEL
LIN {X 0,Y 214.441,Z 497.748,A -85,B 0,C 180,E1 -20878.122,E2 -20878.122} C_VEL
LIN {X 0,Y 214.549,Z 497.753,A -85,B 0,C 180,E1 -20880,E2 -20880} C_VEL
LIN {X 0,Y 214.441,Z 497.764,A -85,B 0,C 180,E1 -20881.878,E2 -20881.878} C_VEL
LIN {X 0,Y 214.194,Z 497.804,A -85,B 0,C 180,E1 -20887.542,E2 -20887.542} C_VEL
LIN {X 0,Y 213.995,Z 497.806,A -85,B 0,C 180,E1 -20891.365,E2 -20891.365} C_VEL
LIN {X 0,Y 213.929,Z 497.833,A -85,B 0,C 180,E1 -20895.237,E2 -20895.237} C_VEL
LIN {X 0,Y 213.834,Z 497.803,A -85,B 0,C 180,E1 -20899.188,E2 -20899.188} C_VEL
LIN {X 0,Y 213.843,Z 497.849,A -85,B 0,C 180,E1 -20903.227,E2 -20903.227} C_VEL
LIN {X 0,Y 213.826,Z 497.818,A -85,B 0,C 180,E1 -20907.45,E2 -20907.45} C_VEL
LIN {X 0,Y 213.774,Z 497.841,A -85,B 0,C 180,E1 -20911.737,E2 -20911.737} C_VEL
LIN {X 0,Y 213.741,Z 497.858,A -85,B 0,C 180,E1 -20916.289,E2 -20916.289} C_VEL
LIN {X 0,Y 213.773,Z 498.027,A -85,B 0,C 180,E1 -20919.3,E2 -20919.3} C_VEL
LIN {X 0,Y 216.742,Z 507.912,A -85,B 0,C 180,E1 -20924.002,E2 -20924.002} C_VEL
LIN {X 0,Y 219.036,Z 516.352,A -85,B 0,C 180,E1 -20927.64,E2 -20927.64} C_VEL
LIN {X 0,Y 220.225,Z 521.387,A -85,B 0,C 180,E1 -20929.669,E2 -20929.669} C_VEL
LIN {X 0,Y 220.685,Z 523.904,A -85,B 0,C 180,E1 -20930.435,E2 -20930.435} C_VEL
LIN {X 0,Y 221.273,Z 528.689,A -85,B 0,C 180,E1 -20931.314,E2 -20931.314} C_VEL
LIN {X 0,Y 221.752,Z 534.138,A -85,B 0,C 180,E1 -20931.923,E2 -20931.923} C_VEL
LIN {X 0,Y 222.34,Z 542.135,A -85,B 0,C 180,E1 -20932.481,E2 -20932.481} C_VEL
LIN {X 0,Y 223.072,Z 550.231,A -85,B 0,C 180,E1 -20932.938,E2 -20932.938} C_VEL
LIN {X 0,Y 225.963,Z 577.289,A -85,B 0,C 180,E1 -20934.499,E2 -20934.499} C_VEL
LIN {X 0,Y 228.314,Z 609.032,A -85,B 0,C 180,E1 -20936.078,E2 -20936.078} C_VEL
LIN {X 0,Y 228.22,Z 616.542,A -85,B 0,C 180,E1 -20936.338,E2 -20936.338} C_VEL
LIN {X 0,Y 227.066,Z 639.794,A -85,B 0,C 180,E1 -20937.093,E2 -20937.093} C_VEL
LIN {X 0,Y 225.632,Z 653.45,A -85,B 0,C 180,E1 -20937.868,E2 -20937.868} C_VEL
LIN {X 0,Y 223.713,Z 665.767,A -85,B 0,C 180,E1 -20938.911,E2 -20938.911} C_VEL
LIN {X 0,Y 221.223,Z 677.5,A -85,B 0,C 180,E1 -20940.239,E2 -20940.239} C_VEL
LIN {X 0,Y 218.382,Z 688.857,A -85,B 0,C 180,E1 -20941.923,E2 -20941.923} C_VEL
LIN {X 0,Y 215.494,Z 699.124,A -85,B 0,C 180,E1 -20943.879,E2 -20943.879} C_VEL
LIN {X 0,Y 212.744,Z 708.41,A -85,B 0,C 180,E1 -20946.13,E2 -20946.13} C_VEL
LIN {X 0,Y 210.086,Z 717.52,A -85,B 0,C 180,E1 -20948.924,E2 -20948.924} C_VEL
LIN {X 0,Y 207.837,Z 724.727,A -85,B 0,C 180,E1 -20951.709,E2 -20951.709} C_VEL
LIN {X 0,Y 206.692,Z 729.914,A -85,B 0,C 180,E1 -20954.216,E2 -20954.216} C_VEL
LIN {X 0,Y 205.762,Z 734.85,A -85,B 0,C 180,E1 -20957.173,E2 -20957.173} C_VEL
LIN {X 0,Y 205.399,Z 738.678,A -85,B 0,C 180,E1 -20960.15,E2 -20960.15} C_VEL
LIN {X 0,Y 205.537,Z 741.05,A -85,B 0,C 180,E1 -20962.573,E2 -20962.573} C_VEL
LIN {X 0,Y 206.088,Z 743.349,A -85,B 0,C 180,E1 -20966.089,E2 -20966.089} C_VEL
LIN {X 0,Y 206.981,Z 744.353,A -85,B 0,C 180,E1 -20970,E2 -20970} C_VEL
LIN {X 0,Y 206.108,Z 743.334,A -85,B 0,C 180,E1 -20973.91,E2 -20973.91} C_VEL
LIN {X 0,Y 205.548,Z 741.001,A -85,B 0,C 180,E1 -20977.451,E2 -20977.451} C_VEL
LIN {X 0,Y 205.461,Z 737.481,A -85,B 0,C 180,E1 -20980.844,E2 -20980.844} C_VEL
LIN {X 0,Y 205.993,Z 733.271,A -85,B 0,C 180,E1 -20983.817,E2 -20983.817} C_VEL
LIN {X 0,Y 207.393,Z 726.893,A -85,B 0,C 180,E1 -20987.248,E2 -20987.248} C_VEL
LIN {X 0,Y 209.314,Z 720.013,A -85,B 0,C 180,E1 -20990.13,E2 -20990.13} C_VEL
LIN {X 0,Y 211.783,Z 711.531,A -85,B 0,C 180,E1 -20992.949,E2 -20992.949} C_VEL
LIN {X 0,Y 214.398,Z 702.888,A -85,B 0,C 180,E1 -20995.222,E2 -20995.222} C_VEL
LIN {X 0,Y 217.422,Z 692.258,A -85,B 0,C 180,E1 -20997.426,E2 -20997.426} C_VEL
LIN {X 0,Y 220.208,Z 681.784,A -85,B 0,C 180,E1 -20999.124,E2 -20999.124} C_VEL
LIN {X 0,Y 222.764,Z 670.3,A -85,B 0,C 180,E1 -21000.578,E2 -21000.578} C_VEL
LIN {X 0,Y 224.749,Z 658.46,A -85,B 0,C 180,E1 -21001.717,E2 -21001.717} C_VEL
LIN {X 0,Y 226.547,Z 644.726,A -85,B 0,C 180,E1 -21002.625,E2 -21002.625} C_VEL
LIN {X 0,Y 227.5,Z 631.402,A -85,B 0,C 180,E1 -21003.177,E2 -21003.177} C_VEL
LIN {X 0,Y 228.261,Z 609.977,A -85,B 0,C 180,E1 -21003.839,E2 -21003.839} C_VEL
LIN {X 0,Y 225.706,Z 575.804,A -85,B 0,C 180,E1 -21005.542,E2 -21005.542} C_VEL
LIN {X 0,Y 222.573,Z 546.888,A -85,B 0,C 180,E1 -21007.223,E2 -21007.223} C_VEL
LIN {X 0,Y 222.114,Z 544.119,A -85,B 0,C 180,E1 -21007.419,E2 -21007.419} C_VEL
LIN {X 0,Y 217.441,Z 533.322,A -85,B 0,C 180,E1 -21008.772,E2 -21008.772} C_VEL
LIN {X 0,Y 213.926,Z 525.28,A -85,B 0,C 180,E1 -21009.909,E2 -21009.909} C_VEL
LIN {X 0,Y 211.726,Z 516.005,A -85,B 0,C 180,E1 -21013.73,E2 -21013.73} C_VEL
LIN {X 0,Y 209.255,Z 507.153,A -85,B 0,C 180,E1 -21017.8,E2 -21017.8} C_VEL
LIN {X 0,Y 206.721,Z 498.825,A -85,B 0,C 180,E1 -21022.108,E2 -21022.108} C_VEL
LIN {X 0,Y 206.699,Z 498.714,A -85,B 0,C 180,E1 -21027.042,E2 -21027.042} C_VEL
LIN {X 0,Y 206.763,Z 498.7,A -85,B 0,C 180,E1 -21032.096,E2 -21032.096} C_VEL
LIN {X 0,Y 206.782,Z 498.729,A -85,B 0,C 180,E1 -21036.584,E2 -21036.584} C_VEL
LIN {X 0,Y 206.869,Z 498.675,A -85,B 0,C 180,E1 -21042.196,E2 -21042.196} C_VEL
LIN {X 0,Y 206.891,Z 498.712,A -85,B 0,C 180,E1 -21046.244,E2 -21046.244} C_VEL
LIN {X 0,Y 207.095,Z 498.672,A -85,B 0,C 180,E1 -21050.231,E2 -21050.231} C_VEL
LIN {X 0,Y 207.057,Z 498.677,A -85,B 0,C 180,E1 -21054.156,E2 -21054.156} C_VEL
LIN {X 0,Y 207.377,Z 498.649,A -85,B 0,C 180,E1 -21058.058,E2 -21058.058} C_VEL
LIN {X 0,Y 207.514,Z 498.633,A -85,B 0,C 180,E1 -21060,E2 -21060} C_VEL
LIN {X 0,Y 207.378,Z 498.63,A -85,B 0,C 180,E1 -21061.942,E2 -21061.942} C_VEL
LIN {X 0,Y 207.136,Z 498.668,A -85,B 0,C 180,E1 -21067.8,E2 -21067.8} C_VEL
LIN {X 0,Y 206.92,Z 498.704,A -85,B 0,C 180,E1 -21071.759,E2 -21071.759} C_VEL
LIN {X 0,Y 206.859,Z 498.695,A -85,B 0,C 180,E1 -21075.772,E2 -21075.772} C_VEL
LIN {X 0,Y 206.774,Z 498.728,A -85,B 0,C 180,E1 -21079.87,E2 -21079.87} C_VEL
LIN {X 0,Y 206.744,Z 498.723,A -85,B 0,C 180,E1 -21084.075,E2 -21084.075} C_VEL
LIN {X 0,Y 206.734,Z 498.684,A -85,B 0,C 180,E1 -21088.421,E2 -21088.421} C_VEL
LIN {X 0,Y 206.696,Z 498.688,A -85,B 0,C 180,E1 -21092.958,E2 -21092.958} C_VEL
LIN {X 0,Y 206.671,Z 498.71,A -85,B 0,C 180,E1 -21097.742,E2 -21097.742} C_VEL
LIN {X 0,Y 206.636,Z 498.703,A -85,B 0,C 180,E1 -21101.562,E2 -21101.562} C_VEL
LIN {X 0,Y 206.633,Z 498.722,A -85,B 0,C 180,E1 -21105.582,E2 -21105.582} C_VEL
LIN {X 0,Y 206.703,Z 498.919,A -85,B 0,C 180,E1 -21109.079,E2 -21109.079} C_VEL
LIN {X 0,Y 206.953,Z 499.944,A -85,B 0,C 180,E1 -21109.443,E2 -21109.443} C_VEL
LIN {X 0,Y 208.552,Z 502.671,A -85,B 0,C 180,E1 -21109.978,E2 -21109.978} C_VEL
LIN {X 0,Y 209.547,Z 503.88,A -85,B 0,C 180,E1 -21110.268,E2 -21110.268} C_VEL
LIN {X 0,Y 217.427,Z 516.415,A -85,B 0,C 180,E1 -21112.554,E2 -21112.554} C_VEL
LIN {X 0,Y 225.545,Z 530.786,A -85,B 0,C 180,E1 -21114.732,E2 -21114.732} C_VEL
LIN {X 0,Y 231.191,Z 542.436,A -85,B 0,C 180,E1 -21116.185,E2 -21116.185} C_VEL
LIN {X 0,Y 230.219,Z 577.83,A -85,B 0,C 180,E1 -21117.327,E2 -21117.327} C_VEL
LIN {X 0,Y 229.708,Z 590.366,A -85,B 0,C 180,E1 -21117.912,E2 -21117.912} C_VEL
LIN {X 0,Y 228.505,Z 603.624,A -85,B 0,C 180,E1 -21118.864,E2 -21118.864} C_VEL
LIN {X 0,Y 226.95,Z 615.893,A -85,B 0,C 180,E1 -21120.122,E2 -21120.122} C_VEL
LIN {X 0,Y 224.855,Z 627.365,A -85,B 0,C 180,E1 -21121.66,E2 -21121.66} C_VEL
LIN {X 0,Y 222.457,Z 638.097,A -85,B 0,C 180,E1 -21123.498,E2 -21123.498} C_VEL
LIN {X 0,Y 220.131,Z 647.285,A -85,B 0,C 180,E1 -21125.479,E2 -21125.479} C_VEL
LIN {X 0,Y 217.855,Z 655.631,A -85,B 0,C 180,E1 -21127.725,E2 -21127.725} C_VEL
LIN {X 0,Y 215.331,Z 663.738,A -85,B 0,C 180,E1 -21130.456,E2 -21130.456} C_VEL
LIN {X 0,Y 212.916,Z 670.842,A -85,B 0,C 180,E1 -21133.504,E2 -21133.504} C_VEL
LIN {X 0,Y 211.141,Z 676.209,A -85,B 0,C 180,E1 -21136.527,E2 -21136.527} C_VEL
LIN {X 0,Y 209.577,Z 680.096,A -85,B 0,C 180,E1 -21139.372,E2 -21139.372} C_VEL
LIN {X 0,Y 208.383,Z 682.965,A -85,B 0,C 180,E1 -21142.247,E2 -21142.247} C_VEL
LIN {X 0,Y 208.037,Z 684.304,A -85,B 0,C 180,E1 -21144.183,E2 -21144.183} C_VEL
LIN {X 0,Y 207.818,Z 685.251,A -85,B 0,C 180,E1 -21146.122,E2 -21146.122} C_VEL
LIN {X 0,Y 207.472,Z 686.079,A -85,B 0,C 180,E1 -21150,E2 -21150} C_VEL
LIN {X 0,Y 207.815,Z 685.306,A -85,B 0,C 180,E1 -21153.878,E2 -21153.878} C_VEL
LIN {X 0,Y 208.367,Z 683.078,A -85,B 0,C 180,E1 -21157.754,E2 -21157.754} C_VEL
LIN {X 0,Y 209.57,Z 680.249,A -85,B 0,C 180,E1 -21160.628,E2 -21160.628} C_VEL
LIN {X 0,Y 211.116,Z 676.417,A -85,B 0,C 180,E1 -21163.475,E2 -21163.475} C_VEL
LIN {X 0,Y 212.811,Z 671.332,A -85,B 0,C 180,E1 -21166.4,E2 -21166.4} C_VEL
LIN {X 0,Y 214.893,Z 665.294,A -85,B 0,C 180,E1 -21169.089,E2 -21169.089} C_VEL
LIN {X 0,Y 217.395,Z 657.506,A -85,B 0,C 180,E1 -21171.825,E2 -21171.825} C_VEL
LIN {X 0,Y 220.083,Z 647.826,A -85,B 0,C 180,E1 -21174.527,E2 -21174.527} C_VEL
LIN {X 0,Y 222.368,Z 638.774,A -85,B 0,C 180,E1 -21176.514,E2 -21176.514} C_VEL
LIN {X 0,Y 224.827,Z 628.243,A -85,B 0,C 180,E1 -21178.33,E2 -21178.33} C_VEL
LIN {X 0,Y 226.919,Z 616.706,A -85,B 0,C 180,E1 -21179.912,E2 -21179.912} C_VEL
LIN {X 0,Y 228.637,Z 605.397,A -85,B 0,C 180,E1 -21181.078,E2 -21181.078} C_VEL
LIN {X 0,Y 229.631,Z 592.903,A -85,B 0,C 180,E1 -21182.068,E2 -21182.068} C_VEL
LIN {X 0,Y 230.214,Z 579.472,A -85,B 0,C 180,E1 -21182.753,E2 -21182.753} C_VEL
LIN {X 0,Y 231.171,Z 542.28,A -85,B 0,C 180,E1 -21183.974,E2 -21183.974} C_VEL
LIN {X 0,Y 224.536,Z 528.896,A -85,B 0,C 180,E1 -21185.687,E2 -21185.687} C_VEL
LIN {X 0,Y 216.187,Z 514.261,A -85,B 0,C 180,E1 -21187.961,E2 -21187.961} C_VEL
LIN {X 0,Y 211.117,Z 506.536,A -85,B 0,C 180,E1 -21189.418,E2 -21189.418} C_VEL
LIN {X 0,Y 208.958,Z 503.105,A -85,B 0,C 180,E1 -21190.077,E2 -21190.077} C_VEL
LIN {X 0,Y 207.285,Z 500.772,A -85,B 0,C 180,E1 -21190.59,E2 -21190.59} C_VEL
LIN {X 0,Y 206.776,Z 499.213,A -85,B 0,C 180,E1 -21190.944,E2 -21190.944} C_VEL
LIN {X 0,Y 206.641,Z 498.74,A -85,B 0,C 180,E1 -21191.562,E2 -21191.562} C_VEL
LIN {X 0,Y 206.633,Z 498.743,A -85,B 0,C 180,E1 -21195.581,E2 -21195.581} C_VEL
LIN {X 0,Y 206.651,Z 498.693,A -85,B 0,C 180,E1 -21199.746,E2 -21199.746} C_VEL
LIN {X 0,Y 206.697,Z 498.738,A -85,B 0,C 180,E1 -21204.688,E2 -21204.688} C_VEL
LIN {X 0,Y 206.703,Z 498.668,A -85,B 0,C 180,E1 -21209.335,E2 -21209.335} C_VEL
LIN {X 0,Y 206.729,Z 498.728,A -85,B 0,C 180,E1 -21213.771,E2 -21213.771} C_VEL
LIN {X 0,Y 206.734,Z 498.714,A -85,B 0,C 180,E1 -21218.04,E2 -21218.04} C_VEL
LIN {X 0,Y 206.868,Z 498.705,A -85,B 0,C 180,E1 -21222.196,E2 -21222.196} C_VEL
LIN {X 0,Y 206.907,Z 498.709,A -85,B 0,C 180,E1 -21226.245,E2 -21226.245} C_VEL
LIN {X 0,Y 207.101,Z 498.662,A -85,B 0,C 180,E1 -21230.231,E2 -21230.231} C_VEL
LIN {X 0,Y 207.174,Z 498.663,A -85,B 0,C 180,E1 -21232.201,E2 -21232.201} C_VEL
LIN {X 0,Y 207.377,Z 498.627,A -85,B 0,C 180,E1 -21238.058,E2 -21238.058} C_VEL
LIN {X 0,Y 207.514,Z 498.629,A -85,B 0,C 180,E1 -21240,E2 -21240} C_VEL
LIN {X 0,Y 207.377,Z 498.644,A -85,B 0,C 180,E1 -21241.942,E2 -21241.942} C_VEL
LIN {X 0,Y 207.136,Z 498.682,A -85,B 0,C 180,E1 -21247.8,E2 -21247.8} C_VEL
LIN {X 0,Y 206.92,Z 498.688,A -85,B 0,C 180,E1 -21251.759,E2 -21251.759} C_VEL
LIN {X 0,Y 206.863,Z 498.706,A -85,B 0,C 180,E1 -21255.771,E2 -21255.771} C_VEL
LIN {X 0,Y 206.763,Z 498.687,A -85,B 0,C 180,E1 -21259.871,E2 -21259.871} C_VEL
LIN {X 0,Y 206.76,Z 498.725,A -85,B 0,C 180,E1 -21264.073,E2 -21264.073} C_VEL
LIN {X 0,Y 206.741,Z 498.708,A -85,B 0,C 180,E1 -21268.419,E2 -21268.419} C_VEL
LIN {X 0,Y 206.699,Z 498.713,A -85,B 0,C 180,E1 -21272.958,E2 -21272.958} C_VEL
LIN {X 0,Y 206.722,Z 498.871,A -85,B 0,C 180,E1 -21277.892,E2 -21277.892} C_VEL
LIN {X 0,Y 209.426,Z 507.761,A -85,B 0,C 180,E1 -21282.416,E2 -21282.416} C_VEL
LIN {X 0,Y 212.082,Z 517.399,A -85,B 0,C 180,E1 -21286.806,E2 -21286.806} C_VEL
LIN {X 0,Y 213.991,Z 525.429,A -85,B 0,C 180,E1 -21290.056,E2 -21290.056} C_VEL
LIN {X 0,Y 219.511,Z 537.809,A -85,B 0,C 180,E1 -21291.759,E2 -21291.759} C_VEL
LIN {X 0,Y 222.501,Z 545.382,A -85,B 0,C 180,E1 -21292.64,E2 -21292.64} C_VEL
LIN {X 0,Y 223.072,Z 550.231,A -85,B 0,C 180,E1 -21292.938,E2 -21292.938} C_VEL
LIN {X 0,Y 223.215,Z 556.044,A -85,B 0,C 180,E1 -21293.191,E2 -21293.191} C_VEL
LIN {X 0,Y 220.471,Z 577.656,A -85,B 0,C 180,E1 -21293.526,E2 -21293.526} C_VEL
LIN {X 0,Y 220.407,Z 581.584,A -85,B 0,C 180,E1 -21293.668,E2 -21293.668} C_VEL
LIN {X 0,Y 222.472,Z 612.283,A -85,B 0,C 180,E1 -21295.221,E2 -21295.221} C_VEL
LIN {X 0,Y 221.155,Z 638.158,A -85,B 0,C 180,E1 -21296.058,E2 -21296.058} C_VEL
LIN {X 0,Y 219.697,Z 651.672,A -85,B 0,C 180,E1 -21296.821,E2 -21296.821} C_VEL
LIN {X 0,Y 217.807,Z 663.751,A -85,B 0,C 180,E1 -21297.833,E2 -21297.833} C_VEL
LIN {X 0,Y 215.494,Z 674.918,A -85,B 0,C 180,E1 -21299.093,E2 -21299.093} C_VEL
LIN {X 0,Y 212.497,Z 686.56,A -85,B 0,C 180,E1 -21300.803,E2 -21300.803} C_VEL
LIN {X 0,Y 209.369,Z 697.061,A -85,B 0,C 180,E1 -21302.784,E2 -21302.784} C_VEL
LIN {X 0,Y 206.794,Z 705.709,A -85,B 0,C 180,E1 -21304.861,E2 -21304.861} C_VEL
LIN {X 0,Y 204.283,Z 713.718,A -85,B 0,C 180,E1 -21307.23,E2 -21307.23} C_VEL
LIN {X 0,Y 202.042,Z 721.027,A -85,B 0,C 180,E1 -21309.916,E2 -21309.916} C_VEL
LIN {X 0,Y 200.485,Z 725.977,A -85,B 0,C 180,E1 -21312.138,E2 -21312.138} C_VEL
LIN {X 0,Y 199.031,Z 732.335,A -85,B 0,C 180,E1 -21315.69,E2 -21315.69} C_VEL
LIN {X 0,Y 198.439,Z 736.528,A -85,B 0,C 180,E1 -21318.768,E2 -21318.768} C_VEL
LIN {X 0,Y 198.468,Z 740.222,A -85,B 0,C 180,E1 -21322.531,E2 -21322.531} C_VEL
LIN {X 0,Y 198.986,Z 742.348,A -85,B 0,C 180,E1 -21325.949,E2 -21325.949} C_VEL
LIN {X 0,Y 199.935,Z 743.362,A -85,B 0,C 180,E1 -21330,E2 -21330} C_VEL
LIN {X 0,Y 199.006,Z 742.333,A -85,B 0,C 180,E1 -21334.05,E2 -21334.05} C_VEL
LIN {X 0,Y 198.483,Z 740.165,A -85,B 0,C 180,E1 -21337.502,E2 -21337.502} C_VEL
LIN {X 0,Y 198.443,Z 736.475,A -85,B 0,C 180,E1 -21341.232,E2 -21341.232} C_VEL
LIN {X 0,Y 199.036,Z 732.261,A -85,B 0,C 180,E1 -21344.31,E2 -21344.31} C_VEL
LIN {X 0,Y 200.54,Z 725.881,A -85,B 0,C 180,E1 -21347.857,E2 -21347.857} C_VEL
LIN {X 0,Y 202.597,Z 719.003,A -85,B 0,C 180,E1 -21350.828,E2 -21350.828} C_VEL
LIN {X 0,Y 205.209,Z 710.522,A -85,B 0,C 180,E1 -21353.729,E2 -21353.729} C_VEL
LIN {X 0,Y 207.971,Z 701.883,A -85,B 0,C 180,E1 -21356.059,E2 -21356.059} C_VEL
LIN {X 0,Y 211.088,Z 691.247,A -85,B 0,C 180,E1 -21358.322,E2 -21358.322} C_VEL
LIN {X 0,Y 214.356,Z 679.331,A -85,B 0,C 180,E1 -21360.27,E2 -21360.27} C_VEL
LIN {X 0,Y 217.074,Z 667.335,A -85,B 0,C 180,E1 -21361.742,E2 -21361.742} C_VEL
LIN {X 0,Y 218.952,Z 656.149,A -85,B 0,C 180,E1 -21362.796,E2 -21362.796} C_VEL
LIN {X 0,Y 220.648,Z 642.886,A -85,B 0,C 180,E1 -21363.672,E2 -21363.672} C_VEL
LIN {X 0,Y 221.575,Z 629.857,A -85,B 0,C 180,E1 -21364.204,E2 -21364.204} C_VEL
LIN {X 0,Y 222.306,Z 610.46,A -85,B 0,C 180,E1 -21364.817,E2 -21364.817} C_VEL
LIN {X 0,Y 219.933,Z 577.322,A -85,B 0,C 180,E1 -21366.523,E2 -21366.523} C_VEL
LIN {X 0,Y 216.999,Z 549.043,A -85,B 0,C 180,E1 -21368.22,E2 -21368.22} C_VEL
LIN {X 0,Y 216.347,Z 546.269,A -85,B 0,C 180,E1 -21368.465,E2 -21368.465} C_VEL
LIN {X 0,Y 212.596,Z 537.432,A -85,B 0,C 180,E1 -21369.617,E2 -21369.617} C_VEL
LIN {X 0,Y 207.923,Z 527.365,A -85,B 0,C 180,E1 -21371.096,E2 -21371.096} C_VEL
LIN {X 0,Y 206.418,Z 523.697,A -85,B 0,C 180,E1 -21371.731,E2 -21371.731} C_VEL
LIN {X 0,Y 204.11,Z 514.605,A -85,B 0,C 180,E1 -21375.793,E2 -21375.793} C_VEL
LIN {X 0,Y 201.605,Z 506.026,A -85,B 0,C 180,E1 -21380.077,E2 -21380.077} C_VEL
LIN {X 0,Y 199.61,Z 499.678,A -85,B 0,C 180,E1 -21383.676,E2 -21383.676} C_VEL
LIN {X 0,Y 199.698,Z 499.592,A -85,B 0,C 180,E1 -21388.136,E2 -21388.136} C_VEL
LIN {X 0,Y 199.683,Z 499.578,A -85,B 0,C 180,E1 -21392.771,E2 -21392.771} C_VEL
LIN {X 0,Y 199.734,Z 499.605,A -85,B 0,C 180,E1 -21397.229,E2 -21397.229} C_VEL
LIN {X 0,Y 199.792,Z 499.552,A -85,B 0,C 180,E1 -21401.758,E2 -21401.758} C_VEL
LIN {X 0,Y 199.832,Z 499.594,A -85,B 0,C 180,E1 -21405.748,E2 -21405.748} C_VEL
LIN {X 0,Y 200.019,Z 499.55,A -85,B 0,C 180,E1 -21409.882,E2 -21409.882} C_VEL
LIN {X 0,Y 200.019,Z 499.555,A -85,B 0,C 180,E1 -21413.949,E2 -21413.949} C_VEL
LIN {X 0,Y 200.317,Z 499.527,A -85,B 0,C 180,E1 -21417.989,E2 -21417.989} C_VEL
LIN {X 0,Y 200.478,Z 499.509,A -85,B 0,C 180,E1 -21420,E2 -21420} C_VEL
LIN {X 0,Y 200.024,Z 499.55,A -85,B 0,C 180,E1 -21424.03,E2 -21424.03} C_VEL
LIN {X 0,Y 200.085,Z 499.542,A -85,B 0,C 180,E1 -21428.077,E2 -21428.077} C_VEL
LIN {X 0,Y 199.869,Z 499.586,A -85,B 0,C 180,E1 -21432.18,E2 -21432.18} C_VEL
LIN {X 0,Y 199.797,Z 499.574,A -85,B 0,C 180,E1 -21436.344,E2 -21436.344} C_VEL
LIN {X 0,Y 199.686,Z 499.603,A -85,B 0,C 180,E1 -21440.607,E2 -21440.607} C_VEL
LIN {X 0,Y 199.662,Z 499.614,A -85,B 0,C 180,E1 -21444.986,E2 -21444.986} C_VEL
LIN {X 0,Y 199.661,Z 499.548,A -85,B 0,C 180,E1 -21449.525,E2 -21449.525} C_VEL
LIN {X 0,Y 199.668,Z 499.552,A -85,B 0,C 180,E1 -21452.356,E2 -21452.356} C_VEL
LIN {X 0,Y 199.618,Z 499.608,A -85,B 0,C 180,E1 -21456.765,E2 -21456.765} C_VEL
LIN {X 0,Y 199.596,Z 499.572,A -85,B 0,C 180,E1 -21459.331,E2 -21459.331} C_VEL
LIN {X 0,Y 199.57,Z 499.593,A -85,B 0,C 180,E1 -21462.31,E2 -21462.31} C_VEL
LIN {X 0,Y 199.629,Z 499.768,A -85,B 0,C 180,E1 -21467.251,E2 -21467.251} C_VEL
LIN {X 0,Y 199.885,Z 500.873,A -85,B 0,C 180,E1 -21467.67,E2 -21467.67} C_VEL
LIN {X 0,Y 201.358,Z 503.466,A -85,B 0,C 180,E1 -21468.209,E2 -21468.209} C_VEL
LIN {X 0,Y 202.698,Z 504.981,A -85,B 0,C 180,E1 -21468.63,E2 -21468.63} C_VEL
LIN {X 0,Y 205.074,Z 508.484,A -85,B 0,C 180,E1 -21469.394,E2 -21469.394} C_VEL
LIN {X 0,Y 212.667,Z 520.65,A -85,B 0,C 180,E1 -21471.709,E2 -21471.709} C_VEL
LIN {X 0,Y 220.398,Z 534.455,A -85,B 0,C 180,E1 -21473.89,E2 -21473.89} C_VEL
LIN {X 0,Y 225.245,Z 544.46,A -85,B 0,C 180,E1 -21475.204,E2 -21475.204} C_VEL
LIN {X 0,Y 224.058,Z 585.731,A -85,B 0,C 180,E1 -21476.643,E2 -21476.643} C_VEL
LIN {X 0,Y 223.141,Z 599.172,A -85,B 0,C 180,E1 -21477.486,E2 -21477.486} C_VEL
LIN {X 0,Y 221.716,Z 611.55,A -85,B 0,C 180,E1 -21478.613,E2 -21478.613} C_VEL
LIN {X 0,Y 219.858,Z 622.904,A -85,B 0,C 180,E1 -21479.999,E2 -21479.999} C_VEL
LIN {X 0,Y 217.609,Z 633.079,A -85,B 0,C 180,E1 -21481.552,E2 -21481.552} C_VEL
LIN {X 0,Y 215.071,Z 643.392,A -85,B 0,C 180,E1 -21483.563,E2 -21483.563} C_VEL
LIN {X 0,Y 212.75,Z 651.801,A -85,B 0,C 180,E1 -21485.612,E2 -21485.612} C_VEL
LIN {X 0,Y 210.455,Z 659.526,A -85,B 0,C 180,E1 -21487.934,E2 -21487.934} C_VEL
LIN {X 0,Y 207.855,Z 667.192,A -85,B 0,C 180,E1 -21490.803,E2 -21490.803} C_VEL
LIN {X 0,Y 205.818,Z 672.936,A -85,B 0,C 180,E1 -21493.533,E2 -21493.533} C_VEL
LIN {X 0,Y 204.313,Z 677.198,A -85,B 0,C 180,E1 -21496.067,E2 -21496.067} C_VEL
LIN {X 0,Y 202.674,Z 681.085,A -85,B 0,C 180,E1 -21499.005,E2 -21499.005} C_VEL
LIN {X 0,Y 201.419,Z 683.954,A -85,B 0,C 180,E1 -21501.977,E2 -21501.977} C_VEL
LIN {X 0,Y 201.045,Z 685.293,A -85,B 0,C 180,E1 -21503.98,E2 -21503.98} C_VEL
LIN {X 0,Y 200.808,Z 686.239,A -85,B 0,C 180,E1 -21505.986,E2 -21505.986} C_VEL
LIN {X 0,Y 200.444,Z 687.067,A -85,B 0,C 180,E1 -21510,E2 -21510} C_VEL
LIN {X 0,Y 200.805,Z 686.294,A -85,B 0,C 180,E1 -21514.014,E2 -21514.014} C_VEL
LIN {X 0,Y 201.402,Z 684.066,A -85,B 0,C 180,E1 -21518.023,E2 -21518.023} C_VEL
LIN {X 0,Y 202.667,Z 681.237,A -85,B 0,C 180,E1 -21520.995,E2 -21520.995} C_VEL
LIN {X 0,Y 204.288,Z 677.404,A -85,B 0,C 180,E1 -21523.934,E2 -21523.934} C_VEL
LIN {X 0,Y 206.078,Z 672.318,A -85,B 0,C 180,E1 -21526.952,E2 -21526.952} C_VEL
LIN {X 0,Y 208.264,Z 666.28,A -85,B 0,C 180,E1 -21529.721,E2 -21529.721} C_VEL
LIN {X 0,Y 210.887,Z 658.491,A -85,B 0,C 180,E1 -21532.534,E2 -21532.534} C_VEL
LIN {X 0,Y 213.707,Z 648.811,A -85,B 0,C 180,E1 -21535.31,E2 -21535.31} C_VEL
LIN {X 0,Y 216.115,Z 639.756,A -85,B 0,C 180,E1 -21537.344,E2 -21537.344} C_VEL
LIN {X 0,Y 218.666,Z 629.226,A -85,B 0,C 180,E1 -21539.204,E2 -21539.204} C_VEL
LIN {X 0,Y 220.893,Z 617.531,A -85,B 0,C 180,E1 -21540.839,E2 -21540.839} C_VEL
LIN {X 0,Y 222.689,Z 606.033,A -85,B 0,C 180,E1 -21542.044,E2 -21542.044} C_VEL
LIN {X 0,Y 223.723,Z 593.738,A -85,B 0,C 180,E1 -21543.031,E2 -21543.031} C_VEL
LIN {X 0,Y 224.357,Z 581.66,A -85,B 0,C 180,E1 -21543.665,E2 -21543.665} C_VEL
LIN {X 0,Y 225.249,Z 548.041,A -85,B 0,C 180,E1 -21544.812,E2 -21544.812} C_VEL
LIN {X 0,Y 225.281,Z 544.403,A -85,B 0,C 180,E1 -21544.946,E2 -21544.946} C_VEL
LIN {X 0,Y 218.628,Z 531.193,A -85,B 0,C 180,E1 -21546.754,E2 -21546.754} C_VEL
LIN {X 0,Y 211.639,Z 518.861,A -85,B 0,C 180,E1 -21548.763,E2 -21548.763} C_VEL
LIN {X 0,Y 204.615,Z 508.001,A -85,B 0,C 180,E1 -21550.918,E2 -21550.918} C_VEL
LIN {X 0,Y 202.114,Z 504.212,A -85,B 0,C 180,E1 -21551.736,E2 -21551.736} C_VEL
LIN {X 0,Y 200.301,Z 501.963,A -85,B 0,C 180,E1 -21552.325,E2 -21552.325} C_VEL
LIN {X 0,Y 199.668,Z 500.08,A -85,B 0,C 180,E1 -21552.757,E2 -21552.757} C_VEL
LIN {X 0,Y 199.573,Z 499.627,A -85,B 0,C 180,E1 -21553.3,E2 -21553.3} C_VEL
LIN {X 0,Y 199.575,Z 499.59,A -85,B 0,C 180,E1 -21558.003,E2 -21558.003} C_VEL
LIN {X 0,Y 199.598,Z 499.572,A -85,B 0,C 180,E1 -21560.77,E2 -21560.77} C_VEL
LIN {X 0,Y 199.612,Z 499.622,A -85,B 0,C 180,E1 -21564.074,E2 -21564.074} C_VEL
LIN {X 0,Y 199.69,Z 499.545,A -85,B 0,C 180,E1 -21568.135,E2 -21568.135} C_VEL
LIN {X 0,Y 199.682,Z 499.585,A -85,B 0,C 180,E1 -21572.771,E2 -21572.771} C_VEL
LIN {X 0,Y 199.71,Z 499.588,A -85,B 0,C 180,E1 -21577.226,E2 -21577.226} C_VEL
LIN {X 0,Y 199.792,Z 499.591,A -85,B 0,C 180,E1 -21581.758,E2 -21581.758} C_VEL
LIN {X 0,Y 199.841,Z 499.582,A -85,B 0,C 180,E1 -21585.749,E2 -21585.749} C_VEL
LIN {X 0,Y 200.067,Z 499.539,A -85,B 0,C 180,E1 -21589.884,E2 -21589.884} C_VEL
LIN {X 0,Y 200.033,Z 499.565,A -85,B 0,C 180,E1 -21593.95,E2 -21593.95} C_VEL
LIN {X 0,Y 200.317,Z 499.505,A -85,B 0,C 180,E1 -21597.989,E2 -21597.989} C_VEL
LIN {X 0,Y 200.478,Z 499.505,A -85,B 0,C 180,E1 -21600,E2 -21600} C_VEL
LIN {X 0,Y 200.022,Z 499.541,A -85,B 0,C 180,E1 -21604.03,E2 -21604.03} C_VEL
LIN {X 0,Y 200.085,Z 499.559,A -85,B 0,C 180,E1 -21608.077,E2 -21608.077} C_VEL
LIN {X 0,Y 199.87,Z 499.569,A -85,B 0,C 180,E1 -21612.18,E2 -21612.18} C_VEL
LIN {X 0,Y 199.8,Z 499.573,A -85,B 0,C 180,E1 -21616.344,E2 -21616.344} C_VEL
LIN {X 0,Y 199.686,Z 499.575,A -85,B 0,C 180,E1 -21620.607,E2 -21620.607} C_VEL
LIN {X 0,Y 199.733,Z 499.603,A -85,B 0,C 180,E1 -21623.817,E2 -21623.817} C_VEL
LIN {X 0,Y 199.71,Z 499.583,A -85,B 0,C 180,E1 -21628.387,E2 -21628.387} C_VEL
LIN {X 0,Y 199.675,Z 499.59,A -85,B 0,C 180,E1 -21632.359,E2 -21632.359} C_VEL
LIN {X 0,Y 199.642,Z 499.777,A -85,B 0,C 180,E1 -21636.38,E2 -21636.38} C_VEL
LIN {X 0,Y 201.628,Z 506.2,A -85,B 0,C 180,E1 -21639.931,E2 -21639.931} C_VEL
LIN {X 0,Y 203.81,Z 513.498,A -85,B 0,C 180,E1 -21643.604,E2 -21643.604} C_VEL
LIN {X 0,Y 205.976,Z 521.74,A -85,B 0,C 180,E1 -21647.399,E2 -21647.399} C_VEL
LIN {X 0,Y 206.547,Z 524.138,A -85,B 0,C 180,E1 -21648.31,E2 -21648.31} C_VEL
LIN {X 0,Y 212.184,Z 536.406,A -85,B 0,C 180,E1 -21650.178,E2 -21650.178} C_VEL
LIN {X 0,Y 216.89,Z 547.549,A -85,B 0,C 180,E1 -21651.629,E2 -21651.629} C_VEL
LIN {X 0,Y 219.881,Z 575.379,A -85,B 0,C 180,E1 -21653.326,E2 -21653.326} C_VEL
LIN {X 0,Y 220.407,Z 581.584,A -85,B 0,C 180,E1 -21653.668,E2 -21653.668} C_VEL
LIN {X 0,Y 220.157,Z 587.454,A -85,B 0,C 180,E1 -21653.851,E2 -21653.851} C_VEL
LIN {X 0,Y 217.117,Z 605.043,A -85,B 0,C 180,E1 -21653.983,E2 -21653.983} C_VEL
LIN {X 0,Y 216.584,Z 610.924,A -85,B 0,C 180,E1 -21654.117,E2 -21654.117} C_VEL
LIN {X 0,Y 216.582,Z 612.878,A -85,B 0,C 180,E1 -21654.194,E2 -21654.194} C_VEL
LIN {X 0,Y 215.274,Z 637.184,A -85,B 0,C 180,E1 -21654.999,E2 -21654.999} C_VEL
LIN {X 0,Y 213.777,Z 650.834,A -85,B 0,C 180,E1 -21655.791,E2 -21655.791} C_VEL
LIN {X 0,Y 211.612,Z 663.772,A -85,B 0,C 180,E1 -21656.914,E2 -21656.914} C_VEL
LIN {X 0,Y 209.023,Z 675.514,A -85,B 0,C 180,E1 -21658.308,E2 -21658.308} C_VEL
LIN {X 0,Y 205.947,Z 686.866,A -85,B 0,C 180,E1 -21660.062,E2 -21660.062} C_VEL
LIN {X 0,Y 202.725,Z 697.115,A -85,B 0,C 180,E1 -21662.095,E2 -21662.095} C_VEL
LIN {X 0,Y 199.778,Z 706.409,A -85,B 0,C 180,E1 -21664.473,E2 -21664.473} C_VEL
LIN {X 0,Y 196.774,Z 715.508,A -85,B 0,C 180,E1 -21667.422,E2 -21667.422} C_VEL
LIN {X 0,Y 194.747,Z 721.593,A -85,B 0,C 180,E1 -21669.887,E2 -21669.887} C_VEL
LIN {X 0,Y 192.905,Z 727.897,A -85,B 0,C 180,E1 -21673.055,E2 -21673.055} C_VEL
LIN {X 0,Y 191.792,Z 732.834,A -85,B 0,C 180,E1 -21676.221,E2 -21676.221} C_VEL
LIN {X 0,Y 191.323,Z 736.669,A -85,B 0,C 180,E1 -21679.417,E2 -21679.417} C_VEL
LIN {X 0,Y 191.421,Z 739.36,A -85,B 0,C 180,E1 -21682.439,E2 -21682.439} C_VEL
LIN {X 0,Y 191.887,Z 741.348,A -85,B 0,C 180,E1 -21685.799,E2 -21685.799} C_VEL
LIN {X 0,Y 192.889,Z 742.371,A -85,B 0,C 180,E1 -21690,E2 -21690} C_VEL
LIN {X 0,Y 191.907,Z 741.332,A -85,B 0,C 180,E1 -21694.2,E2 -21694.2} C_VEL
LIN {X 0,Y 191.432,Z 739.309,A -85,B 0,C 180,E1 -21697.586,E2 -21697.586} C_VEL
LIN {X 0,Y 191.418,Z 735.466,A -85,B 0,C 180,E1 -21701.65,E2 -21701.65} C_VEL
LIN {X 0,Y 192.098,Z 731.252,A -85,B 0,C 180,E1 -21704.838,E2 -21704.838} C_VEL
LIN {X 0,Y 193.717,Z 724.869,A -85,B 0,C 180,E1 -21708.508,E2 -21708.508} C_VEL
LIN {X 0,Y 195.926,Z 717.995,A -85,B 0,C 180,E1 -21711.572,E2 -21711.572} C_VEL
LIN {X 0,Y 198.685,Z 709.515,A -85,B 0,C 180,E1 -21714.558,E2 -21714.558} C_VEL
LIN {X 0,Y 201.582,Z 700.876,A -85,B 0,C 180,E1 -21716.951,E2 -21716.951} C_VEL
LIN {X 0,Y 204.832,Z 690.24,A -85,B 0,C 180,E1 -21719.27,E2 -21719.27} C_VEL
LIN {X 0,Y 207.853,Z 679.768,A -85,B 0,C 180,E1 -21721.039,E2 -21721.039} C_VEL
LIN {X 0,Y 210.653,Z 668.29,A -85,B 0,C 180,E1 -21722.545,E2 -21722.545} C_VEL
LIN {X 0,Y 212.799,Z 656.447,A -85,B 0,C 180,E1 -21723.728,E2 -21723.728} C_VEL
LIN {X 0,Y 214.687,Z 642.642,A -85,B 0,C 180,E1 -21724.679,E2 -21724.679} C_VEL
LIN {X 0,Y 215.674,Z 629.903,A -85,B 0,C 180,E1 -21725.234,E2 -21725.234} C_VEL
LIN {X 0,Y 216.455,Z 611.831,A -85,B 0,C 180,E1 -21725.806,E2 -21725.806} C_VEL
LIN {X 0,Y 214.127,Z 577.789,A -85,B 0,C 180,E1 -21727.621,E2 -21727.621} C_VEL
LIN {X 0,Y 211.348,Z 550.175,A -85,B 0,C 180,E1 -21729.345,E2 -21729.345} C_VEL
LIN {X 0,Y 206.429,Z 538.271,A -85,B 0,C 180,E1 -21730.96,E2 -21730.96} C_VEL
LIN {X 0,Y 200.779,Z 526.525,A -85,B 0,C 180,E1 -21732.874,E2 -21732.874} C_VEL
LIN {X 0,Y 198.911,Z 522.319,A -85,B 0,C 180,E1 -21733.68,E2 -21733.68} C_VEL
LIN {X 0,Y 196.581,Z 513.612,A -85,B 0,C 180,E1 -21737.875,E2 -21737.875} C_VEL
LIN {X 0,Y 194.26,Z 505.898,A -85,B 0,C 180,E1 -21742.046,E2 -21742.046} C_VEL
LIN {X 0,Y 192.572,Z 500.551,A -85,B 0,C 180,E1 -21745.312,E2 -21745.312} C_VEL
LIN {X 0,Y 192.603,Z 500.492,A -85,B 0,C 180,E1 -21749.279,E2 -21749.279} C_VEL
LIN {X 0,Y 192.662,Z 500.458,A -85,B 0,C 180,E1 -21751.691,E2 -21751.691} C_VEL
LIN {X 0,Y 192.702,Z 500.48,A -85,B 0,C 180,E1 -21756.348,E2 -21756.348} C_VEL
LIN {X 0,Y 192.727,Z 500.43,A -85,B 0,C 180,E1 -21761.458,E2 -21761.458} C_VEL
LIN {X 0,Y 192.76,Z 500.475,A -85,B 0,C 180,E1 -21765.213,E2 -21765.213} C_VEL
LIN {X 0,Y 192.941,Z 500.429,A -85,B 0,C 180,E1 -21769.566,E2 -21769.566} C_VEL
LIN {X 0,Y 192.981,Z 500.434,A -85,B 0,C 180,E1 -21773.728,E2 -21773.728} C_VEL
LIN {X 0,Y 193.258,Z 500.404,A -85,B 0,C 180,E1 -21777.916,E2 -21777.916} C_VEL
LIN {X 0,Y 193.442,Z 500.385,A -85,B 0,C 180,E1 -21780,E2 -21780} C_VEL
LIN {X 0,Y 192.97,Z 500.43,A -85,B 0,C 180,E1 -21784.177,E2 -21784.177} C_VEL
LIN {X 0,Y 193.032,Z 500.418,A -85,B 0,C 180,E1 -21788.374,E2 -21788.374} C_VEL
LIN {X 0,Y 192.797,Z 500.469,A -85,B 0,C 180,E1 -21792.634,E2 -21792.634} C_VEL
LIN {X 0,Y 192.752,Z 500.454,A -85,B 0,C 180,E1 -21796.959,E2 -21796.959} C_VEL
LIN {X 0,Y 192.617,Z 500.474,A -85,B 0,C 180,E1 -21801.4,E2 -21801.4} C_VEL
LIN {X 0,Y 192.644,Z 500.48,A -85,B 0,C 180,E1 -21804.214,E2 -21804.214} C_VEL
LIN {X 0,Y 192.641,Z 500.428,A -85,B 0,C 180,E1 -21808.889,E2 -21808.889} C_VEL
LIN {X 0,Y 192.594,Z 500.444,A -85,B 0,C 180,E1 -21813.187,E2 -21813.187} C_VEL
LIN {X 0,Y 192.582,Z 500.486,A -85,B 0,C 180,E1 -21816.598,E2 -21816.598} C_VEL
LIN {X 0,Y 192.507,Z 500.456,A -85,B 0,C 180,E1 -21821.082,E2 -21821.082} C_VEL
LIN {X 0,Y 192.588,Z 500.739,A -85,B 0,C 180,E1 -21825.326,E2 -21825.326} C_VEL
LIN {X 0,Y 192.894,Z 501.958,A -85,B 0,C 180,E1 -21825.738,E2 -21825.738} C_VEL
LIN {X 0,Y 194.364,Z 504.427,A -85,B 0,C 180,E1 -21826.318,E2 -21826.318} C_VEL
LIN {X 0,Y 195.633,Z 505.732,A -85,B 0,C 180,E1 -21826.75,E2 -21826.75} C_VEL
LIN {X 0,Y 197.877,Z 509.213,A -85,B 0,C 180,E1 -21827.551,E2 -21827.551} C_VEL
LIN {X 0,Y 204.181,Z 518.725,A -85,B 0,C 180,E1 -21829.643,E2 -21829.643} C_VEL
LIN {X 0,Y 210.635,Z 529.479,A -85,B 0,C 180,E1 -21831.637,E2 -21831.637} C_VEL
LIN {X 0,Y 217.873,Z 543.402,A -85,B 0,C 180,E1 -21833.75,E2 -21833.75} C_VEL
LIN {X 0,Y 219.438,Z 546.748,A -85,B 0,C 180,E1 -21834.194,E2 -21834.194} C_VEL
LIN {X 0,Y 218.199,Z 586.872,A -85,B 0,C 180,E1 -21835.632,E2 -21835.632} C_VEL
LIN {X 0,Y 217.237,Z 600.239,A -85,B 0,C 180,E1 -21836.494,E2 -21836.494} C_VEL
LIN {X 0,Y 215.747,Z 612.545,A -85,B 0,C 180,E1 -21837.641,E2 -21837.641} C_VEL
LIN {X 0,Y 213.837,Z 623.702,A -85,B 0,C 180,E1 -21839.029,E2 -21839.029} C_VEL
LIN {X 0,Y 211.456,Z 634.071,A -85,B 0,C 180,E1 -21840.645,E2 -21840.645} C_VEL
LIN {X 0,Y 208.8,Z 644.384,A -85,B 0,C 180,E1 -21842.704,E2 -21842.704} C_VEL
LIN {X 0,Y 206.369,Z 652.793,A -85,B 0,C 180,E1 -21844.806,E2 -21844.806} C_VEL
LIN {X 0,Y 203.959,Z 660.517,A -85,B 0,C 180,E1 -21847.192,E2 -21847.192} C_VEL
LIN {X 0,Y 201.231,Z 668.182,A -85,B 0,C 180,E1 -21850.145,E2 -21850.145} C_VEL
LIN {X 0,Y 199.088,Z 673.925,A -85,B 0,C 180,E1 -21852.96,E2 -21852.96} C_VEL
